  MoveL (T16970) to (106.02, 107.35, 18.1) mm, rotated rx 180 ry 0 rz -180 deg; joints [2.549, 70.013, -35.529, 4.496, -34.567, -3.705]
  Call Extruder 0.1339
  MoveL (T16971) to (109.55, 103.82, 18.1) mm, rotated rx 180 ry 0 rz -180 deg; joints [2.138, 71.113, -37.597, 3.868, -33.577, -3.224]
  Call Extruder 0.01361
  MoveL (T16972) to (109.04, 103.82, 18.1) mm, rotated rx 180 ry 0 rz -180 deg; joints [2.138, 71.113, -37.597, 3.868, -33.577, -3.224]
  Call Extruder 0.11544
  MoveL (T16973) to (106, 106.86, 18.1) mm, rotated rx 180 ry 0 rz -180 deg; joints [2.138, 71.113, -37.597, 3.868, -33.577, -3.224]
  Call Extruder 0.01361
  MoveL (T16974) to (106, 106.35, 18.1) mm, rotated rx 180 ry 0 rz -180 deg; joints [2.086, 71.108, -37.586, 3.773, -33.579, -3.145]
  Call Extruder 0.09619
  MoveL (T16975) to (108.53, 103.82, 18.1) mm, rotated rx 180 ry 0 rz -180 deg; joints [2.086, 71.108, -37.586, 3.773, -33.579, -3.145]
  Call Extruder 0.01361
  MoveL (T16976) to (108.03, 103.82, 18.1) mm, rotated rx 180 ry 0 rz -180 deg; joints [2.086, 71.108, -37.586, 3.773, -33.579, -3.145]
  Call Extruder 0.07694
  MoveL (T16977) to (106, 105.85, 18.1) mm, rotated rx 180 ry 0 rz -180 deg; joints [2.523, 69.937, -35.386, 4.443, -34.632, -3.658]
  Call Extruder 0.01361
  MoveL (T16978) to (106, 105.34, 18.1) mm, rotated rx 180 ry 0 rz -180 deg; joints [2.523, 69.937, -35.386, 4.443, -34.632, -3.658]
  Call Extruder 0.06379
  MoveL (T16979) to (107.68, 103.66, 18.1) mm, rotated rx 180 ry 0 rz -180 deg; joints [2.519, 69.932, -35.375, 4.435, -34.636, -3.651]
  Set speed (45.0 mm/s)
  Call Extruder -1.6
  MoveL (T16980) to (107.68, 103.66, 18.1) mm, rotated rx 180 ry 0 rz -180 deg; joints [2.519, 69.932, -35.375, 4.435, -34.636, -3.651]
  Set speed (120.0 mm/s)
  MoveL (T16981) to (107.68, 103.66, 18.1) mm, rotated rx 180 ry 0 rz -180 deg; joints [2.519, 69.932, -35.375, 4.435, -34.636, -3.651]
  Call Extruder -0.38
  MoveL (T16982) to (106.93, 104.41, 18.1) mm, rotated rx 180 ry 0 rz -180 deg; joints [2.519, 69.932, -35.375, 4.435, -34.636, -3.651]
  Set speed (45.0 mm/s)
  Call Extruder -0.02
  MoveL (T16983) to (106.93, 104.41, 18.1) mm, rotated rx 180 ry 0 rz -180 deg; joints [2.472, 69.926, -35.365, 4.353, -34.639, -3.583]
  Set speed (150.0 mm/s)
  MoveL (T16984) to (106.93, 104.41, 20.1) mm, rotated rx 180 ry 0 rz -180 deg; joints [2.472, 69.926, -35.365, 4.353, -34.639, -3.583]
  MoveL (T16985) to (108.68, 114.32, 20.1) mm, rotated rx 180 ry 0 rz -180 deg; joints [2.033, 71.102, -37.575, 3.678, -33.581, -3.065]
  MoveL (T16986) to (108.68, 114.32, 18.1) mm, rotated rx 180 ry 0 rz -180 deg; joints [2.033, 71.102, -37.575, 3.678, -33.581, -3.065]
  Set speed (40.0 mm/s)
  Call Extruder 2.0
  MoveL (T16987) to (108.68, 114.32, 18.1) mm, rotated rx 180 ry 0 rz -180 deg; joints [1.981, 71.097, -37.565, 3.582, -33.583, -2.986]
  Set speed (25.0 mm/s)
  MoveL (T16988) to (108.68, 114.32, 18.1) mm, rotated rx 180 ry 0 rz -180 deg; joints [1.981, 71.097, -37.565, 3.582, -33.583, -2.986]
  Call Extruder 0.09856
  MoveL (T16989) to (106.08, 116.92, 18.1) mm, rotated rx 180 ry 0 rz -180 deg; joints [1.981, 71.097, -37.565, 3.582, -33.583, -2.986]
  Call Extruder 0.01361
  MoveL (T16990) to (106.08, 116.41, 18.1) mm, rotated rx 180 ry 0 rz -180 deg; joints [1.981, 71.097, -37.565, 3.582, -33.583, -2.986]
  Call Extruder 0.07931
  MoveL (T16991) to (108.17, 114.32, 18.1) mm, rotated rx 180 ry 0 rz -180 deg; joints [2.42, 69.919, -35.353, 4.259, -34.641, -3.506]
  Set speed (45.0 mm/s)
  Call Extruder -1.6
  MoveL (T16992) to (108.17, 114.32, 18.1) mm, rotated rx 180 ry 0 rz -180 deg; joints [2.42, 69.919, -35.353, 4.259, -34.641, -3.506]
  Set speed (120.0 mm/s)
  MoveL (T16993) to (108.17, 114.32, 18.1) mm, rotated rx 180 ry 0 rz -180 deg; joints [2.42, 69.919, -35.353, 4.259, -34.641, -3.506]
  Call Extruder -0.38
  MoveL (T16994) to (107.42, 115.08, 18.1) mm, rotated rx 180 ry 0 rz -180 deg; joints [2.42, 69.919, -35.353, 4.259, -34.641, -3.506]
  Set speed (45.0 mm/s)
  Call Extruder -0.02
  MoveL (T16995) to (107.42, 115.08, 18.1) mm, rotated rx 180 ry 0 rz -180 deg; joints [2.367, 69.913, -35.341, 4.166, -34.643, -3.429]
  Set speed (150.0 mm/s)
  MoveL (T16996) to (107.42, 115.08, 20.1) mm, rotated rx 180 ry 0 rz -180 deg; joints [2.367, 69.913, -35.341, 4.166, -34.643, -3.429]
  MoveL (T16997) to (109.4, 105.47, 20.1) mm, rotated rx 180 ry 0 rz -180 deg; joints [2.367, 69.913, -35.341, 4.166, -34.643, -3.429]
  MoveL (T16998) to (109.4, 105.47, 18.3) mm, rotated rx 180 ry 0 rz -180 deg; joints [2.367, 69.913, -35.341, 4.166, -34.643, -3.429]
  Set speed (40.0 mm/s)
  Call Extruder 2.0
  MoveL (T16999) to (109.4, 105.47, 18.3) mm, rotated rx 180 ry 0 rz -180 deg; joints [1.928, 71.091, -37.555, 3.487, -33.585, -2.906]
  Set speed (31.5 mm/s)
  MoveL (T17000) to (109.4, 105.47, 18.3) mm, rotated rx 180 ry 0 rz -180 deg; joints [1.928, 71.091, -37.555, 3.487, -33.585, -2.906]
  Call Extruder 0.25145
  MoveL (T17001) to (117.65, 105.47, 18.3) mm, rotated rx 180 ry 0 rz -180 deg; joints [1.876, 71.086, -37.545, 3.392, -33.587, -2.827]
  Call Extruder 0.10939
  MoveL (T17002) to (117.65, 109.06, 18.3) mm, rotated rx 180 ry 0 rz -180 deg; joints [1.876, 71.086, -37.545, 3.392, -33.587, -2.827]
  Call Extruder 0.14732
  MoveL (T17003) to (112.81, 109.06, 18.3) mm, rotated rx 180 ry 0 rz -180 deg; joints [1.876, 71.086, -37.545, 3.392, -33.587, -2.827]
  Call Extruder 0.31102
  MoveL (T17004) to (117.47, 118.15, 18.3) mm, rotated rx 180 ry 0 rz -180 deg; joints [2.314, 69.907, -35.33, 4.072, -34.645, -3.352]
  Call Extruder 0.05209
  MoveL (T17005) to (117.47, 119.86, 18.3) mm, rotated rx 180 ry 0 rz -180 deg; joints [2.314, 69.907, -35.33, 4.072, -34.645, -3.352]
  Call Extruder 0.29244
  MoveL (T17006) to (107.87, 119.86, 18.3) mm, rotated rx 180 ry 0 rz -180 deg; joints [2.314, 69.907, -35.33, 4.072, -34.645, -3.352]
  Call Extruder 0.10939
  MoveL (T17007) to (107.87, 116.27, 18.3) mm, rotated rx 180 ry 0 rz -180 deg; joints [2.314, 69.907, -35.33, 4.072, -34.645, -3.352]
  Call Extruder 0.13869
  MoveL (T17008) to (112.42, 116.27, 18.3) mm, rotated rx 180 ry 0 rz -180 deg; joints [2.261, 69.902, -35.319, 3.979, -34.647, -3.275]
  Call Extruder 0.31084
  MoveL (T17009) to (107.78, 107.18, 18.3) mm, rotated rx 180 ry 0 rz -180 deg; joints [2.261, 69.902, -35.319, 3.979, -34.647, -3.275]
  Call Extruder 0.05206
  MoveL (T17010) to (107.78, 105.47, 18.3) mm, rotated rx 180 ry 0 rz -180 deg; joints [1.826, 71.072, -37.519, 3.302, -33.597, -2.751]
  Call Extruder 0.04735
  MoveL (T17011) to (109.34, 105.47, 18.3) mm, rotated rx 180 ry 0 rz -180 deg; joints [1.826, 71.072, -37.519, 3.302, -33.597, -2.751]
  Set speed (150.0 mm/s)
  MoveL (T17012) to (109, 105.88, 18.3) mm, rotated rx 180 ry 0 rz -180 deg; joints [1.826, 71.072, -37.519, 3.302, -33.597, -2.751]
  Set speed (31.5 mm/s)
  MoveL (T17013) to (109, 105.88, 18.3) mm, rotated rx 180 ry 0 rz -180 deg; joints [1.828, 70.917, -37.227, 3.293, -33.734, -2.74]
  Call Extruder 0.25124
  MoveL (T17014) to (117.24, 105.88, 18.3) mm, rotated rx 180 ry 0 rz -180 deg; joints [1.828, 70.917, -37.227, 3.293, -33.734, -2.74]
  Call Extruder 0.08459
  MoveL (T17015) to (117.24, 108.65, 18.3) mm, rotated rx 180 ry 0 rz -180 deg; joints [1.828, 70.917, -37.227, 3.293, -33.734, -2.74]
  Call Extruder 0.1552
  MoveL (T17016) to (112.15, 108.65, 18.3) mm, rotated rx 180 ry 0 rz -180 deg; joints [1.828, 70.917, -37.227, 3.293, -33.734, -2.74]
  Call Extruder 0.32831
  MoveL (T17017) to (117.06, 118.25, 18.3) mm, rotated rx 180 ry 0 rz -180 deg; joints [2.208, 69.896, -35.308, 3.886, -34.649, -3.198]
  Call Extruder 0.0367
  MoveL (T17018) to (117.06, 119.45, 18.3) mm, rotated rx 180 ry 0 rz -180 deg; joints [2.208, 69.896, -35.308, 3.886, -34.649, -3.198]
  Call Extruder 0.26763
  MoveL (T17019) to (108.27, 119.45, 18.3) mm, rotated rx 180 ry 0 rz -180 deg; joints [2.155, 69.89, -35.298, 3.793, -34.651, -3.121]
  Call Extruder 0.08459
  MoveL (T17020) to (108.27, 116.67, 18.3) mm, rotated rx 180 ry 0 rz -180 deg; joints [2.155, 69.89, -35.298, 3.793, -34.651, -3.121]
  Call Extruder 0.14654
  MoveL (T17021) to (113.08, 116.67, 18.3) mm, rotated rx 180 ry 0 rz -180 deg; joints [1.83, 70.762, -36.936, 3.284, -33.87, -2.728]
  Call Extruder 0.32811
  MoveL (T17022) to (108.19, 107.08, 18.3) mm, rotated rx 180 ry 0 rz -180 deg; joints [1.83, 70.762, -36.936, 3.284, -33.87, -2.728]
  Call Extruder 0.03668
  MoveL (T17023) to (108.19, 105.88, 18.3) mm, rotated rx 180 ry 0 rz -180 deg; joints [1.831, 70.608, -36.647, 3.276, -34.005, -2.717]
  Call Extruder 0.02276
  MoveL (T17024) to (108.94, 105.88, 18.3) mm, rotated rx 180 ry 0 rz -180 deg; joints [1.831, 70.608, -36.647, 3.276, -34.005, -2.717]
  Set speed (150.0 mm/s)
  MoveL (T17025) to (108.6, 106.28, 18.3) mm, rotated rx 180 ry 0 rz -180 deg; joints [1.831, 70.608, -36.647, 3.276, -34.005, -2.717]
  Set speed (25.0 mm/s)
  MoveL (T17026) to (108.6, 106.28, 18.3) mm, rotated rx 180 ry 0 rz -180 deg; joints [2.103, 69.885, -35.287, 3.699, -34.653, -3.045]
  Call Extruder 0.25102
  MoveL (T17027) to (116.84, 106.28, 18.3) mm, rotated rx 180 ry 0 rz -180 deg; joints [2.103, 69.885, -35.287, 3.699, -34.653, -3.045]
  Call Extruder 0.05979
  MoveL (T17028) to (116.84, 108.25, 18.3) mm, rotated rx 180 ry 0 rz -180 deg; joints [2.103, 69.885, -35.287, 3.699, -34.653, -3.045]
  Call Extruder 0.16307
  MoveL (T17029) to (111.48, 108.25, 18.3) mm, rotated rx 180 ry 0 rz -180 deg; joints [2.053, 69.88, -35.278, 3.612, -34.655, -2.972]
  Call Extruder 0.3456
  MoveL (T17030) to (116.65, 118.34, 18.3) mm, rotated rx 180 ry 0 rz -180 deg; joints [2.053, 69.88, -35.278, 3.612, -34.655, -2.972]
  Call Extruder 0.02131
  MoveL (T17031) to (116.65, 119.04, 18.3) mm, rotated rx 180 ry 0 rz -180 deg; joints [2.053, 69.88, -35.278, 3.612, -34.655, -2.972]
  Call Extruder 0.24283
  MoveL (T17032) to (108.68, 119.04, 18.3) mm, rotated rx 180 ry 0 rz -180 deg; joints [2.053, 69.88, -35.278, 3.612, -34.655, -2.972]
  Call Extruder 0.05979
  MoveL (T17033) to (108.68, 117.08, 18.3) mm, rotated rx 180 ry 0 rz -180 deg; joints [2.047, 69.886, -35.289, 3.602, -34.649, -2.965]
  Call Extruder 0.15438
  MoveL (T17034) to (113.75, 117.08, 18.3) mm, rotated rx 180 ry 0 rz -180 deg; joints [2.047, 69.886, -35.289, 3.602, -34.649, -2.965]
  Call Extruder 0.34538
  MoveL (T17035) to (108.6, 106.98, 18.3) mm, rotated rx 180 ry 0 rz -180 deg; joints [1.816, 70.502, -36.447, 3.241, -34.097, -2.685]
  Call Extruder 0.01947
  MoveL (T17036) to (108.6, 106.34, 18.3) mm, rotated rx 180 ry 0 rz -180 deg; joints [1.816, 70.502, -36.447, 3.241, -34.097, -2.685]
  Set speed (150.0 mm/s)
  MoveL (T17037) to (108.54, 105.89, 18.3) mm, rotated rx 180 ry 0 rz -180 deg; joints [1.816, 70.502, -36.447, 3.241, -34.097, -2.685]
  Set speed (45.0 mm/s)
  Call Extruder -1.6
  MoveL (T17038) to (108.54, 105.89, 18.3) mm, rotated rx 180 ry 0 rz -180 deg; joints [1.816, 70.502, -36.447, 3.241, -34.097, -2.685]
  Set speed (120.0 mm/s)
  MoveL (T17039) to (108.54, 105.89, 18.3) mm, rotated rx 180 ry 0 rz -180 deg; joints [1.816, 70.502, -36.447, 3.241, -34.097, -2.685]
  Call Extruder -0.38
  MoveL (T17040) to (109.66, 106.33, 18.3) mm, rotated rx 180 ry 0 rz -180 deg; joints [1.816, 70.502, -36.447, 3.241, -34.097, -2.685]
  Set speed (45.0 mm/s)
  Call Extruder -0.02
  MoveL (T17041) to (109.66, 106.33, 18.3) mm, rotated rx 180 ry 0 rz -180 deg; joints [1.816, 70.502, -36.447, 3.241, -34.097, -2.685]
  Set speed (150.0 mm/s)
  MoveL (T17042) to (109.66, 106.33, 20.3) mm, rotated rx 180 ry 0 rz -180 deg; joints [1.816, 70.502, -36.447, 3.241, -34.097, -2.685]
  MoveL (T17043) to (104.34, 103.54, 20.3) mm, rotated rx 180 ry 0 rz -180 deg; joints [1.816, 70.502, -36.447, 3.241, -34.097, -2.685]
  MoveL (T17044) to (104.34, 103.54, 18.3) mm, rotated rx 180 ry 0 rz -180 deg; joints [1.816, 70.502, -36.447, 3.241, -34.097, -2.685]
  Set speed (40.0 mm/s)
  Call Extruder 2.0
  MoveL (T17045) to (104.34, 103.54, 18.3) mm, rotated rx 180 ry 0 rz -180 deg; joints [1.816, 70.502, -36.447, 3.241, -34.097, -2.685]
  Set speed (31.5 mm/s)
  MoveL (T17046) to (104.34, 103.54, 18.3) mm, rotated rx 180 ry 0 rz -180 deg; joints [1.816, 70.502, -36.447, 3.241, -34.097, -2.685]
  Call Extruder 0.52159
  MoveL (T17047) to (121.46, 103.54, 18.3) mm, rotated rx 180 ry 0 rz -180 deg; joints [1.898, 70.28, -36.031, 3.37, -34.296, -2.785]
  Call Extruder 0.54596
  MoveL (T17048) to (121.46, 121.46, 18.3) mm, rotated rx 180 ry 0 rz -180 deg; joints [1.898, 70.28, -36.031, 3.37, -34.296, -2.785]
  Call Extruder 0.54596
  MoveL (T17049) to (103.54, 121.46, 18.3) mm, rotated rx 180 ry 0 rz -180 deg; joints [1.898, 70.28, -36.031, 3.37, -34.296, -2.785]
  Call Extruder 0.54596
  MoveL (T17050) to (103.54, 103.54, 18.3) mm, rotated rx 180 ry 0 rz -180 deg; joints [1.898, 70.28, -36.031, 3.37, -34.296, -2.785]
  Call Extruder 0.02254
  MoveL (T17051) to (104.28, 103.54, 18.3) mm, rotated rx 180 ry 0 rz -180 deg; joints [1.898, 70.28, -36.031, 3.37, -34.296, -2.785]
  Set speed (150.0 mm/s)
  MoveL (T17052) to (103.53, 103.13, 18.3) mm, rotated rx 180 ry 0 rz -180 deg; joints [1.898, 70.28, -36.031, 3.37, -34.296, -2.785]
  Set speed (31.5 mm/s)
  MoveL (T17053) to (103.53, 103.13, 18.3) mm, rotated rx 180 ry 0 rz -180 deg; joints [1.898, 70.28, -36.031, 3.37, -34.296, -2.785]
  Call Extruder 0.55858
  MoveL (T17054) to (121.87, 103.13, 18.3) mm, rotated rx 180 ry 0 rz -180 deg; joints [1.586, 70.545, -36.923, 2.863, -33.655, -2.384]
  Call Extruder 0.57077
  MoveL (T17055) to (121.87, 121.87, 18.3) mm, rotated rx 180 ry 0 rz -180 deg; joints [1.586, 70.778, -36.966, 2.849, -33.845, -2.367]
  Call Extruder 0.57077
  MoveL (T17056) to (103.13, 121.87, 18.3) mm, rotated rx 180 ry 0 rz -180 deg; joints [1.586, 70.778, -36.966, 2.849, -33.845, -2.367]
  Call Extruder 0.57077
  MoveL (T17057) to (103.13, 103.13, 18.3) mm, rotated rx 180 ry 0 rz -180 deg; joints [1.586, 70.778, -36.966, 2.849, -33.845, -2.367]
  Call Extruder 0.01036
  MoveL (T17058) to (103.47, 103.13, 18.3) mm, rotated rx 180 ry 0 rz -180 deg; joints [1.586, 70.778, -36.966, 2.849, -33.845, -2.367]
  Set speed (150.0 mm/s)
  MoveL (T17059) to (102.72, 102.81, 18.3) mm, rotated rx 180 ry 0 rz -180 deg; joints [1.586, 70.778, -36.966, 2.849, -33.845, -2.367]
  Set speed (25.0 mm/s)
  MoveL (T17060) to (102.72, 102.81, 18.3) mm, rotated rx 180 ry 0 rz -180 deg; joints [1.586, 70.778, -36.966, 2.849, -33.845, -2.367]
  Call Extruder 0.00259
  MoveL (T17061) to (102.72, 102.72, 18.3) mm, rotated rx 180 ry 0 rz -180 deg; joints [1.586, 70.778, -36.966, 2.849, -33.845, -2.367]
  Call Extruder 0.59557
  MoveL (T17062) to (122.28, 102.72, 18.3) mm, rotated rx 180 ry 0 rz -180 deg; joints [1.586, 70.778, -36.966, 2.849, -33.845, -2.367]
  Call Extruder 0.59557
  MoveL (T17063) to (122.28, 122.28, 18.3) mm, rotated rx 180 ry 0 rz -180 deg; joints [1.816, 70.153, -35.791, 3.215, -34.404, -2.654]
  Call Extruder 0.59557
  MoveL (T17064) to (102.72, 122.28, 18.3) mm, rotated rx 180 ry 0 rz -180 deg; joints [1.816, 70.153, -35.791, 3.215, -34.404, -2.654]
  Call Extruder 0.59115
  MoveL (T17065) to (102.72, 102.87, 18.3) mm, rotated rx 180 ry 0 rz -180 deg; joints [1.816, 70.153, -35.791, 3.215, -34.404, -2.654]
  Set speed (150.0 mm/s)
  MoveL (T17066) to (102.78, 102.75, 18.3) mm, rotated rx 180 ry 0 rz -180 deg; joints [1.816, 70.153, -35.791, 3.215, -34.404, -2.654]
  Set speed (45.0 mm/s)
  Call Extruder -1.6
  MoveL (T17067) to (102.78, 102.75, 18.3) mm, rotated rx 180 ry 0 rz -180 deg; joints [1.819, 70.136, -35.759, 3.219, -34.419, -2.656]
  Set speed (120.0 mm/s)
  MoveL (T17068) to (102.78, 102.75, 18.3) mm, rotated rx 180 ry 0 rz -180 deg; joints [1.819, 70.136, -35.759, 3.219, -34.419, -2.656]
  Call Extruder -0.05166
  MoveL (T17069) to (102.72, 102.72, 18.3) mm, rotated rx 180 ry 0 rz -180 deg; joints [1.819, 70.136, -35.759, 3.219, -34.419, -2.656]
  Call Extruder -0.32834
  MoveL (T17070) to (103.65, 102.72, 18.3) mm, rotated rx 180 ry 0 rz -180 deg; joints [1.82, 69.997, -35.498, 3.211, -34.541, -2.646]
  Set speed (45.0 mm/s)
  Call Extruder -0.02
  MoveL (T17071) to (103.65, 102.72, 18.3) mm, rotated rx 180 ry 0 rz -180 deg; joints [1.82, 69.997, -35.498, 3.211, -34.541, -2.646]
  Set speed (150.0 mm/s)
  MoveL (T17072) to (103.65, 102.72, 20.3) mm, rotated rx 180 ry 0 rz -180 deg; joints [1.551, 70.727, -36.87, 2.782, -33.888, -2.31]
  MoveL (T17073) to (106.29, 103.84, 20.3) mm, rotated rx 180 ry 0 rz -180 deg; joints [1.551, 70.727, -36.87, 2.782, -33.888, -2.31]
  MoveL (T17074) to (106.29, 103.84, 18.3) mm, rotated rx 180 ry 0 rz -180 deg; joints [1.551, 70.727, -36.87, 2.782, -33.888, -2.31]
  Set speed (40.0 mm/s)
  Call Extruder 2.0
  MoveL (T17075) to (106.29, 103.84, 18.3) mm, rotated rx 180 ry 0 rz -180 deg; joints [1.499, 70.723, -36.863, 2.688, -33.889, -2.232]
  Set speed (31.5 mm/s)
  MoveL (T17076) to (106.29, 103.84, 18.3) mm, rotated rx 180 ry 0 rz -180 deg; joints [1.499, 70.723, -36.863, 2.688, -33.889, -2.232]
  Call Extruder 0.07441
  MoveL (T17077) to (103.84, 103.84, 18.3) mm, rotated rx 180 ry 0 rz -180 deg; joints [1.822, 69.849, -35.221, 3.204, -34.67, -2.636]
  Call Extruder 0.16673
  MoveL (T17078) to (107.71, 107.71, 18.3) mm, rotated rx 180 ry 0 rz -180 deg; joints [1.822, 69.849, -35.221, 3.204, -34.67, -2.636]
  Call Extruder 0.00815
  MoveL (T17079) to (107.84, 107.95, 18.3) mm, rotated rx 180 ry 0 rz -180 deg; joints [1.823, 69.702, -34.944, 3.196, -34.8, -2.625]
  Call Extruder 0.17197
  MoveL (T17080) to (103.84, 111.94, 18.3) mm, rotated rx 180 ry 0 rz -180 deg; joints [1.823, 69.702, -34.944, 3.196, -34.8, -2.625]
  Call Extruder 0.03385
  MoveL (T17081) to (103.84, 113.06, 18.3) mm, rotated rx 180 ry 0 rz -180 deg; joints [1.823, 69.702, -34.944, 3.196, -34.8, -2.625]
  Call Extruder 0.16015
  MoveL (T17082) to (107.56, 116.77, 18.3) mm, rotated rx 180 ry 0 rz -180 deg; joints [1.446, 70.719, -36.855, 2.594, -33.891, -2.154]
  Call Extruder 0.02027
  MoveL (T17083) to (107.56, 117.44, 18.3) mm, rotated rx 180 ry 0 rz -180 deg; joints [1.446, 70.719, -36.855, 2.594, -33.891, -2.154]
  Call Extruder 0.16015
  MoveL (T17084) to (103.84, 121.16, 18.3) mm, rotated rx 180 ry 0 rz -180 deg; joints [1.395, 70.715, -36.848, 2.503, -33.892, -2.078]
  Call Extruder 0.07441
  MoveL (T17085) to (106.29, 121.16, 18.3) mm, rotated rx 180 ry 0 rz -180 deg; joints [1.395, 70.715, -36.848, 2.503, -33.892, -2.078]
  Set speed (45.0 mm/s)
  Call Extruder -1.6
  MoveL (T17086) to (106.29, 121.16, 18.3) mm, rotated rx 180 ry 0 rz -180 deg; joints [1.395, 70.715, -36.848, 2.503, -33.892, -2.078]
  Set speed (120.0 mm/s)
  MoveL (T17087) to (106.29, 121.16, 18.3) mm, rotated rx 180 ry 0 rz -180 deg; joints [1.395, 70.711, -36.84, 2.503, -33.896, -2.078]
  Call Extruder -0.38
  MoveL (T17088) to (105.22, 121.16, 18.3) mm, rotated rx 180 ry 0 rz -180 deg; joints [1.395, 70.711, -36.84, 2.503, -33.896, -2.078]
  Set speed (45.0 mm/s)
  Call Extruder -0.02
  MoveL (T17089) to (105.22, 121.16, 18.3) mm, rotated rx 180 ry 0 rz -180 deg; joints [1.825, 69.556, -34.67, 3.189, -34.928, -2.615]
  Set speed (150.0 mm/s)
  MoveL (T17090) to (105.22, 121.16, 20.3) mm, rotated rx 180 ry 0 rz -180 deg; joints [1.827, 69.411, -34.398, 3.182, -35.055, -2.605]
  MoveL (T17091) to (109.84, 111.88, 20.3) mm, rotated rx 180 ry 0 rz -180 deg; joints [1.827, 69.411, -34.398, 3.182, -35.055, -2.605]
  MoveL (T17092) to (109.84, 111.88, 18.3) mm, rotated rx 180 ry 0 rz -180 deg; joints [1.827, 69.411, -34.398, 3.182, -35.055, -2.605]
  Set speed (40.0 mm/s)
  Call Extruder 2.0
  MoveL (T17093) to (109.84, 111.88, 18.3) mm, rotated rx 180 ry 0 rz -180 deg; joints [1.397, 70.559, -36.554, 2.496, -34.03, -2.069]
  Set speed (31.5 mm/s)
  MoveL (T17094) to (109.84, 111.88, 18.3) mm, rotated rx 180 ry 0 rz -180 deg; joints [1.397, 70.559, -36.554, 2.496, -34.03, -2.069]
  Call Extruder 0.07441
  MoveL (T17095) to (110.95, 114.05, 18.3) mm, rotated rx 180 ry 0 rz -180 deg; joints [1.397, 70.559, -36.554, 2.496, -34.03, -2.069]
  Call Extruder 0.08223
  MoveL (T17096) to (109.04, 115.96, 18.3) mm, rotated rx 180 ry 0 rz -180 deg; joints [1.398, 70.407, -36.269, 2.49, -34.163, -2.061]
  Call Extruder 0.07057
  MoveL (T17097) to (111.36, 115.96, 18.3) mm, rotated rx 180 ry 0 rz -180 deg; joints [1.398, 70.407, -36.269, 2.49, -34.163, -2.061]
  Call Extruder 0.32359
  MoveL (T17098) to (103.84, 108.45, 18.3) mm, rotated rx 180 ry 0 rz -180 deg; joints [1.829, 69.267, -34.127, 3.175, -35.182, -2.596]
  Call Extruder 0.03385
  MoveL (T17099) to (103.84, 107.34, 18.3) mm, rotated rx 180 ry 0 rz -180 deg; joints [1.829, 69.267, -34.127, 3.175, -35.182, -2.596]
  Call Extruder 0.15054
  MoveL (T17100) to (107.34, 103.84, 18.3) mm, rotated rx 180 ry 0 rz -180 deg; joints [1.83, 69.124, -33.858, 3.168, -35.308, -2.586]
  Call Extruder 0.03385
  MoveL (T17101) to (108.45, 103.84, 18.3) mm, rotated rx 180 ry 0 rz -180 deg; joints [1.83, 69.124, -33.858, 3.168, -35.308, -2.586]
  Call Extruder 0.05679
  MoveL (T17102) to (109.77, 105.16, 18.3) mm, rotated rx 180 ry 0 rz -180 deg; joints [1.83, 69.124, -33.858, 3.168, -35.308, -2.586]
  Call Extruder 0.02614
  MoveL (T17103) to (110.63, 105.16, 18.3) mm, rotated rx 180 ry 0 rz -180 deg; joints [1.83, 69.124, -33.858, 3.168, -35.308, -2.586]
  Call Extruder 0.05679
  MoveL (T17104) to (111.94, 103.84, 18.3) mm, rotated rx 180 ry 0 rz -180 deg; joints [1.399, 70.257, -35.986, 2.484, -34.295, -2.053]
  Call Extruder 0.03385
  MoveL (T17105) to (113.06, 103.84, 18.3) mm, rotated rx 180 ry 0 rz -180 deg; joints [1.399, 70.257, -35.986, 2.484, -34.295, -2.053]
  Call Extruder 0.05679
  MoveL (T17106) to (114.37, 105.16, 18.3) mm, rotated rx 180 ry 0 rz -180 deg; joints [1.399, 70.257, -35.986, 2.484, -34.295, -2.053]
  Call Extruder 0.02614
  MoveL (T17107) to (115.23, 105.16, 18.3) mm, rotated rx 180 ry 0 rz -180 deg; joints [1.401, 70.107, -35.706, 2.478, -34.427, -2.044]
  Call Extruder 0.05679
  MoveL (T17108) to (116.55, 103.84, 18.3) mm, rotated rx 180 ry 0 rz -180 deg; joints [1.401, 70.107, -35.706, 2.478, -34.427, -2.044]
  Call Extruder 0.03385
  MoveL (T17109) to (117.66, 103.84, 18.3) mm, rotated rx 180 ry 0 rz -180 deg; joints [1.832, 68.981, -33.59, 3.161, -35.433, -2.576]
  Call Extruder 0.15054
  MoveL (T17110) to (121.16, 107.34, 18.3) mm, rotated rx 180 ry 0 rz -180 deg; joints [1.832, 68.981, -33.59, 3.161, -35.433, -2.576]
  Call Extruder 0.03385
  MoveL (T17111) to (121.16, 108.45, 18.3) mm, rotated rx 180 ry 0 rz -180 deg; joints [1.834, 68.84, -33.323, 3.154, -35.557, -2.567]
  Call Extruder 0.23679
  MoveL (T17112) to (115.66, 113.95, 18.3) mm, rotated rx 180 ry 0 rz -180 deg; joints [1.402, 69.958, -35.426, 2.472, -34.557, -2.036]
  Call Extruder 0.10426
  MoveL (T17113) to (114.1, 110.9, 18.3) mm, rotated rx 180 ry 0 rz -180 deg; joints [1.402, 69.958, -35.426, 2.472, -34.557, -2.036]
  Call Extruder 0.06615
  MoveL (T17114) to (115.64, 109.36, 18.3) mm, rotated rx 180 ry 0 rz -180 deg; joints [1.402, 69.958, -35.426, 2.472, -34.557, -2.036]
  Call Extruder 0.05076
  MoveL (T17115) to (113.97, 109.36, 18.3) mm, rotated rx 180 ry 0 rz -180 deg; joints [1.403, 69.811, -35.149, 2.466, -34.687, -2.028]
  Call Extruder 0.30958
  MoveL (T17116) to (121.16, 116.55, 18.3) mm, rotated rx 180 ry 0 rz -180 deg; joints [1.403, 69.811, -35.149, 2.466, -34.687, -2.028]
  Call Extruder 0.03385
  MoveL (T17117) to (121.16, 117.66, 18.3) mm, rotated rx 180 ry 0 rz -180 deg; joints [1.403, 69.811, -35.149, 2.466, -34.687, -2.028]
  Call Extruder 0.15054
  MoveL (T17118) to (117.66, 121.16, 18.3) mm, rotated rx 180 ry 0 rz -180 deg; joints [1.814, 68.753, -33.16, 3.114, -35.633, -2.532]
  Call Extruder 0.03385
  MoveL (T17119) to (116.55, 121.16, 18.3) mm, rotated rx 180 ry 0 rz -180 deg; joints [1.814, 68.753, -33.16, 3.114, -35.633, -2.532]
  Call Extruder 0.04278
  MoveL (T17120) to (115.56, 120.16, 18.3) mm, rotated rx 180 ry 0 rz -180 deg; joints [1.814, 68.753, -33.16, 3.114, -35.633, -2.532]
  Call Extruder 0.04595
  MoveL (T17121) to (114.05, 120.16, 18.3) mm, rotated rx 180 ry 0 rz -180 deg; joints [1.814, 68.753, -33.16, 3.114, -35.633, -2.532]
  Call Extruder 0.04278
  MoveL (T17122) to (113.06, 121.16, 18.3) mm, rotated rx 180 ry 0 rz -180 deg; joints [1.788, 68.68, -33.024, 3.065, -35.695, -2.49]
  Call Extruder 0.03385
  MoveL (T17123) to (111.94, 121.16, 18.3) mm, rotated rx 180 ry 0 rz -180 deg; joints [1.788, 68.68, -33.024, 3.065, -35.695, -2.49]
  Call Extruder 0.04278
  MoveL (T17124) to (110.95, 120.16, 18.3) mm, rotated rx 180 ry 0 rz -180 deg; joints [1.788, 68.68, -33.024, 3.065, -35.695, -2.49]
  Call Extruder 0.04595
  MoveL (T17125) to (109.44, 120.16, 18.3) mm, rotated rx 180 ry 0 rz -180 deg; joints [1.788, 68.68, -33.024, 3.065, -35.695, -2.49]
  Call Extruder 0.04278
  MoveL (T17126) to (108.45, 121.16, 18.3) mm, rotated rx 180 ry 0 rz -180 deg; joints [1.404, 69.664, -34.873, 2.46, -34.816, -2.02]
  Call Extruder 0.03385
  MoveL (T17127) to (107.34, 121.16, 18.3) mm, rotated rx 180 ry 0 rz -180 deg; joints [1.404, 69.664, -34.873, 2.46, -34.816, -2.02]
  Call Extruder 0.15054
  MoveL (T17128) to (103.84, 117.66, 18.3) mm, rotated rx 180 ry 0 rz -180 deg; joints [1.406, 69.519, -34.599, 2.455, -34.944, -2.013]
  Call Extruder 0.03385
  MoveL (T17129) to (103.84, 116.55, 18.3) mm, rotated rx 180 ry 0 rz -180 deg; joints [1.406, 69.519, -34.599, 2.455, -34.944, -2.013]
  Call Extruder 0.23899
  MoveL (T17130) to (109.39, 111, 18.3) mm, rotated rx 180 ry 0 rz -180 deg; joints [1.406, 69.519, -34.599, 2.455, -34.944, -2.013]
  Call Extruder 0.07441
  MoveL (T17131) to (108.28, 108.83, 18.3) mm, rotated rx 180 ry 0 rz -180 deg; joints [1.762, 68.608, -32.888, 3.017, -35.757, -2.449]
  Set speed (45.0 mm/s)
  Call Extruder -1.6
  MoveL (T17132) to (108.28, 108.83, 18.3) mm, rotated rx 180 ry 0 rz -180 deg; joints [1.762, 68.608, -32.888, 3.017, -35.757, -2.449]
  Set speed (120.0 mm/s)
  MoveL (T17133) to (108.28, 108.83, 18.3) mm, rotated rx 180 ry 0 rz -180 deg; joints [1.762, 68.608, -32.888, 3.017, -35.757, -2.449]
  Call Extruder -0.38
  MoveL (T17134) to (108.77, 109.78, 18.3) mm, rotated rx 180 ry 0 rz -180 deg; joints [1.737, 68.536, -32.754, 2.968, -35.819, -2.408]
  Set speed (45.0 mm/s)
  Call Extruder -0.02
  MoveL (T17135) to (108.77, 109.78, 18.3) mm, rotated rx 180 ry 0 rz -180 deg; joints [1.737, 68.536, -32.754, 2.968, -35.819, -2.408]
  Set speed (150.0 mm/s)
  MoveL (T17136) to (108.77, 109.78, 20.3) mm, rotated rx 180 ry 0 rz -180 deg; joints [1.737, 68.536, -32.754, 2.968, -35.819, -2.408]
  MoveL (T17137) to (118.71, 103.84, 20.3) mm, rotated rx 180 ry 0 rz -180 deg; joints [1.737, 68.536, -32.754, 2.968, -35.819, -2.408]
  MoveL (T17138) to (118.71, 103.84, 18.3) mm, rotated rx 180 ry 0 rz -180 deg; joints [1.407, 69.374, -34.327, 2.449, -35.071, -2.005]
  Set speed (40.0 mm/s)
  Call Extruder 2.0
  MoveL (T17139) to (118.71, 103.84, 18.3) mm, rotated rx 180 ry 0 rz -180 deg; joints [1.407, 69.374, -34.327, 2.449, -35.071, -2.005]
  Set speed (31.5 mm/s)
  MoveL (T17140) to (118.71, 103.84, 18.3) mm, rotated rx 180 ry 0 rz -180 deg; joints [1.408, 69.23, -34.056, 2.444, -35.198, -1.997]
  Call Extruder 0.07441
  MoveL (T17141) to (121.16, 103.84, 18.3) mm, rotated rx 180 ry 0 rz -180 deg; joints [1.408, 69.23, -34.056, 2.444, -35.198, -1.997]
  Call Extruder 0.13782
  MoveL (T17142) to (117.96, 107.04, 18.3) mm, rotated rx 180 ry 0 rz -180 deg; joints [1.711, 68.464, -32.618, 2.92, -35.881, -2.366]
  Call Extruder 0.05185
  MoveL (T17143) to (117.96, 108.75, 18.3) mm, rotated rx 180 ry 0 rz -180 deg; joints [1.711, 68.464, -32.618, 2.92, -35.881, -2.366]
  Call Extruder 0.13782
  MoveL (T17144) to (121.16, 111.94, 18.3) mm, rotated rx 180 ry 0 rz -180 deg; joints [1.711, 68.464, -32.618, 2.92, -35.881, -2.366]
  Call Extruder 0.03385
  MoveL (T17145) to (121.16, 113.06, 18.3) mm, rotated rx 180 ry 0 rz -180 deg; joints [1.685, 68.393, -32.484, 2.872, -35.943, -2.326]
  Call Extruder 0.16962
  MoveL (T17146) to (117.22, 116.99, 18.3) mm, rotated rx 180 ry 0 rz -180 deg; joints [1.685, 68.393, -32.484, 2.872, -35.943, -2.326]
  Call Extruder 0.01582
  MoveL (T17147) to (117.45, 117.45, 18.3) mm, rotated rx 180 ry 0 rz -180 deg; joints [1.685, 68.393, -32.484, 2.872, -35.943, -2.326]
  Call Extruder 0.15942
  MoveL (T17148) to (121.16, 121.16, 18.3) mm, rotated rx 180 ry 0 rz -180 deg; joints [1.41, 69.087, -33.788, 2.439, -35.324, -1.99]
  Call Extruder 0.07441
  MoveL (T17149) to (118.71, 121.16, 18.3) mm, rotated rx 180 ry 0 rz -180 deg; joints [1.41, 69.087, -33.788, 2.439, -35.324, -1.99]
  Set speed (45.0 mm/s)
  Call Extruder -1.6
  MoveL (T17150) to (118.71, 121.16, 18.3) mm, rotated rx 180 ry 0 rz -180 deg; joints [1.41, 69.087, -33.788, 2.439, -35.324, -1.99]
  Set speed (120.0 mm/s)
  MoveL (T17151) to (118.71, 121.16, 18.3) mm, rotated rx 180 ry 0 rz -180 deg; joints [1.411, 68.944, -33.52, 2.433, -35.448, -1.983]
  Call Extruder -0.38
  MoveL (T17152) to (119.78, 121.16, 18.3) mm, rotated rx 180 ry 0 rz -180 deg; joints [1.411, 68.944, -33.52, 2.433, -35.448, -1.983]
  Set speed (45.0 mm/s)
  Call Extruder -0.02
  MoveL (T17153) to (119.78, 121.16, 18.3) mm, rotated rx 180 ry 0 rz -180 deg; joints [1.846, 67.87, -31.502, 3.11, -36.408, -2.504]
  Set speed (150.0 mm/s)
  MoveL (T17154) to (119.78, 121.16, 20.3) mm, rotated rx 180 ry 0 rz -180 deg; joints [1.846, 67.87, -31.502, 3.11, -36.408, -2.504]
  MoveL (T17155) to (109.4, 105.47, 20.3) mm, rotated rx 180 ry 0 rz -180 deg; joints [1.846, 67.87, -31.502, 3.11, -36.408, -2.504]
  MoveL (T17156) to (109.4, 105.47, 18.5) mm, rotated rx 180 ry 0 rz -180 deg; joints [1.847, 67.735, -31.248, 3.105, -36.527, -2.496]
  Set speed (40.0 mm/s)
  Call Extruder 2.0
  MoveL (T17157) to (109.4, 105.47, 18.5) mm, rotated rx 180 ry 0 rz -180 deg; joints [1.847, 67.735, -31.248, 3.105, -36.527, -2.496]
  Set speed (31.6 mm/s)
  MoveL (T17158) to (109.4, 105.47, 18.5) mm, rotated rx 180 ry 0 rz -180 deg; joints [1.847, 67.735, -31.248, 3.105, -36.527, -2.496]
  Call Extruder 0.25145
  MoveL (T17159) to (117.65, 105.47, 18.5) mm, rotated rx 180 ry 0 rz -180 deg; joints [1.412, 68.803, -33.255, 2.428, -35.573, -1.975]
  Call Extruder 0.10939
  MoveL (T17160) to (117.65, 109.06, 18.5) mm, rotated rx 180 ry 0 rz -180 deg; joints [1.412, 68.803, -33.255, 2.428, -35.573, -1.975]
  Call Extruder 0.14732
  MoveL (T17161) to (112.81, 109.06, 18.5) mm, rotated rx 180 ry 0 rz -180 deg; joints [1.414, 68.662, -32.99, 2.423, -35.696, -1.968]
  Call Extruder 0.31102
  MoveL (T17162) to (117.47, 118.15, 18.5) mm, rotated rx 180 ry 0 rz -180 deg; joints [1.849, 67.6, -30.994, 3.099, -36.646, -2.487]
  Call Extruder 0.05209
  MoveL (T17163) to (117.47, 119.86, 18.5) mm, rotated rx 180 ry 0 rz -180 deg; joints [1.849, 67.6, -30.994, 3.099, -36.646, -2.487]
  Call Extruder 0.29244
  MoveL (T17164) to (107.87, 119.86, 18.5) mm, rotated rx 180 ry 0 rz -180 deg; joints [1.851, 67.465, -30.742, 3.093, -36.764, -2.479]
  Call Extruder 0.10939
  MoveL (T17165) to (107.87, 116.27, 18.5) mm, rotated rx 180 ry 0 rz -180 deg; joints [1.415, 68.522, -32.727, 2.418, -35.819, -1.961]
  Call Extruder 0.13869
  MoveL (T17166) to (112.42, 116.27, 18.5) mm, rotated rx 180 ry 0 rz -180 deg; joints [1.415, 68.522, -32.727, 2.418, -35.819, -1.961]
  Call Extruder 0.31084
  MoveL (T17167) to (107.78, 107.18, 18.5) mm, rotated rx 180 ry 0 rz -180 deg; joints [1.415, 68.522, -32.727, 2.418, -35.819, -1.961]
  Call Extruder 0.05206
  MoveL (T17168) to (107.78, 105.47, 18.5) mm, rotated rx 180 ry 0 rz -180 deg; joints [1.416, 68.383, -32.466, 2.413, -35.941, -1.954]
  Call Extruder 0.04735
  MoveL (T17169) to (109.34, 105.47, 18.5) mm, rotated rx 180 ry 0 rz -180 deg; joints [1.416, 68.383, -32.466, 2.413, -35.941, -1.954]
  Set speed (150.0 mm/s)
  MoveL (T17170) to (109, 105.88, 18.5) mm, rotated rx 180 ry 0 rz -180 deg; joints [1.416, 68.383, -32.466, 2.413, -35.941, -1.954]
  Set speed (31.6 mm/s)
  MoveL (T17171) to (109, 105.88, 18.5) mm, rotated rx 180 ry 0 rz -180 deg; joints [1.416, 68.383, -32.466, 2.413, -35.941, -1.954]
  Call Extruder 0.25124
  MoveL (T17172) to (117.24, 105.88, 18.5) mm, rotated rx 180 ry 0 rz -180 deg; joints [1.852, 67.332, -30.491, 3.088, -36.881, -2.471]
  Call Extruder 0.08459
  MoveL (T17173) to (117.24, 108.65, 18.5) mm, rotated rx 180 ry 0 rz -180 deg; joints [1.852, 67.332, -30.491, 3.088, -36.881, -2.471]
  Call Extruder 0.1552
  MoveL (T17174) to (112.15, 108.65, 18.5) mm, rotated rx 180 ry 0 rz -180 deg; joints [1.852, 67.332, -30.491, 3.088, -36.881, -2.471]
  Call Extruder 0.32831
  MoveL (T17175) to (117.06, 118.25, 18.5) mm, rotated rx 180 ry 0 rz -180 deg; joints [1.852, 67.332, -30.491, 3.088, -36.881, -2.471]
  Call Extruder 0.0367
  MoveL (T17176) to (117.06, 119.45, 18.5) mm, rotated rx 180 ry 0 rz -180 deg; joints [1.854, 67.199, -30.242, 3.082, -36.997, -2.462]
  Call Extruder 0.26763
  MoveL (T17177) to (108.27, 119.45, 18.5) mm, rotated rx 180 ry 0 rz -180 deg; joints [1.854, 67.199, -30.242, 3.082, -36.997, -2.462]
  Call Extruder 0.08459
  MoveL (T17178) to (108.27, 116.67, 18.5) mm, rotated rx 180 ry 0 rz -180 deg; joints [1.854, 67.199, -30.242, 3.082, -36.997, -2.462]
  Call Extruder 0.14654
  MoveL (T17179) to (113.08, 116.67, 18.5) mm, rotated rx 180 ry 0 rz -180 deg; joints [1.854, 67.199, -30.242, 3.082, -36.997, -2.462]
  Call Extruder 0.32811
  MoveL (T17180) to (108.19, 107.08, 18.5) mm, rotated rx 180 ry 0 rz -180 deg; joints [1.417, 68.245, -32.206, 2.408, -36.063, -1.947]
  Call Extruder 0.03668
  MoveL (T17181) to (108.19, 105.88, 18.5) mm, rotated rx 180 ry 0 rz -180 deg; joints [1.417, 68.245, -32.206, 2.408, -36.063, -1.947]
  Call Extruder 0.02276
  MoveL (T17182) to (108.94, 105.88, 18.5) mm, rotated rx 180 ry 0 rz -180 deg; joints [1.419, 68.107, -31.948, 2.404, -36.184, -1.94]
  Set speed (150.0 mm/s)
  MoveL (T17183) to (108.6, 106.28, 18.5) mm, rotated rx 180 ry 0 rz -180 deg; joints [1.419, 68.107, -31.948, 2.404, -36.184, -1.94]
  Set speed (25.0 mm/s)
  MoveL (T17184) to (108.6, 106.28, 18.5) mm, rotated rx 180 ry 0 rz -180 deg; joints [1.419, 68.107, -31.948, 2.404, -36.184, -1.94]
  Call Extruder 0.25102
  MoveL (T17185) to (116.84, 106.28, 18.5) mm, rotated rx 180 ry 0 rz -180 deg; joints [1.856, 67.067, -29.994, 3.077, -37.113, -2.454]
  Call Extruder 0.05979
  MoveL (T17186) to (116.84, 108.25, 18.5) mm, rotated rx 180 ry 0 rz -180 deg; joints [1.856, 67.067, -29.994, 3.077, -37.113, -2.454]
  Call Extruder 0.16307
  MoveL (T17187) to (111.48, 108.25, 18.5) mm, rotated rx 180 ry 0 rz -180 deg; joints [1.856, 67.067, -29.994, 3.077, -37.113, -2.454]
  Call Extruder 0.3456
  MoveL (T17188) to (116.65, 118.34, 18.5) mm, rotated rx 180 ry 0 rz -180 deg; joints [1.858, 66.936, -29.747, 3.071, -37.229, -2.446]
  Call Extruder 0.02131
  MoveL (T17189) to (116.65, 119.04, 18.5) mm, rotated rx 180 ry 0 rz -180 deg; joints [1.858, 66.936, -29.747, 3.071, -37.229, -2.446]
  Call Extruder 0.24283
  MoveL (T17190) to (108.68, 119.04, 18.5) mm, rotated rx 180 ry 0 rz -180 deg; joints [1.858, 66.936, -29.747, 3.071, -37.229, -2.446]
  Call Extruder 0.05979
  MoveL (T17191) to (108.68, 117.08, 18.5) mm, rotated rx 180 ry 0 rz -180 deg; joints [1.42, 67.971, -31.691, 2.399, -36.304, -1.934]
  Call Extruder 0.15438
  MoveL (T17192) to (113.75, 117.08, 18.5) mm, rotated rx 180 ry 0 rz -180 deg; joints [1.42, 67.971, -31.691, 2.399, -36.304, -1.934]
  Call Extruder 0.34538
  MoveL (T17193) to (108.6, 106.98, 18.5) mm, rotated rx 180 ry 0 rz -180 deg; joints [1.42, 67.971, -31.691, 2.399, -36.304, -1.934]
  Call Extruder 0.01947
  MoveL (T17194) to (108.6, 106.34, 18.5) mm, rotated rx 180 ry 0 rz -180 deg; joints [1.42, 67.971, -31.691, 2.399, -36.304, -1.934]
  Set speed (150.0 mm/s)
  MoveL (T17195) to (108.54, 105.89, 18.5) mm, rotated rx 180 ry 0 rz -180 deg; joints [1.421, 67.834, -31.435, 2.394, -36.423, -1.927]
  Set speed (45.0 mm/s)
  Call Extruder -1.6
  MoveL (T17196) to (108.54, 105.89, 18.5) mm, rotated rx 180 ry 0 rz -180 deg; joints [1.421, 67.834, -31.435, 2.394, -36.423, -1.927]
  Set speed (120.0 mm/s)
  MoveL (T17197) to (108.54, 105.89, 18.5) mm, rotated rx 180 ry 0 rz -180 deg; joints [1.858, 66.808, -29.506, 3.064, -37.341, -2.437]
  Call Extruder -0.38
  MoveL (T17198) to (109.66, 106.33, 18.5) mm, rotated rx 180 ry 0 rz -180 deg; joints [1.858, 66.808, -29.506, 3.064, -37.341, -2.437]
  Set speed (45.0 mm/s)
  Call Extruder -0.02
  MoveL (T17199) to (109.66, 106.33, 18.5) mm, rotated rx 180 ry 0 rz -180 deg; joints [1.857, 66.798, -29.489, 3.061, -37.349, -2.434]
  Set speed (150.0 mm/s)
  MoveL (T17200) to (109.66, 106.33, 20.5) mm, rotated rx 180 ry 0 rz -180 deg; joints [1.857, 66.798, -29.489, 3.061, -37.349, -2.434]
  MoveL (T17201) to (104.34, 103.54, 20.5) mm, rotated rx 180 ry 0 rz -180 deg; joints [1.833, 66.738, -29.375, 3.019, -37.401, -2.399]
  MoveL (T17202) to (104.34, 103.54, 18.5) mm, rotated rx 180 ry 0 rz -180 deg; joints [1.833, 66.738, -29.375, 3.019, -37.401, -2.399]
  Set speed (40.0 mm/s)
  Call Extruder 2.0
  MoveL (T17203) to (104.34, 103.54, 18.5) mm, rotated rx 180 ry 0 rz -180 deg; joints [1.423, 67.699, -31.181, 2.39, -36.542, -1.921]
  Set speed (31.6 mm/s)
  MoveL (T17204) to (104.34, 103.54, 18.5) mm, rotated rx 180 ry 0 rz -180 deg; joints [1.423, 67.699, -31.181, 2.39, -36.542, -1.921]
  Call Extruder 0.52159
  MoveL (T17205) to (121.46, 103.54, 18.5) mm, rotated rx 180 ry 0 rz -180 deg; joints [1.423, 67.699, -31.181, 2.39, -36.542, -1.921]
  Call Extruder 0.54596
  MoveL (T17206) to (121.46, 121.46, 18.5) mm, rotated rx 180 ry 0 rz -180 deg; joints [1.424, 67.564, -30.928, 2.386, -36.66, -1.914]
  Call Extruder 0.54596
  MoveL (T17207) to (103.54, 121.46, 18.5) mm, rotated rx 180 ry 0 rz -180 deg; joints [1.424, 67.564, -30.928, 2.386, -36.66, -1.914]
  Call Extruder 0.54596
  MoveL (T17208) to (103.54, 103.54, 18.5) mm, rotated rx 180 ry 0 rz -180 deg; joints [1.424, 67.564, -30.928, 2.386, -36.66, -1.914]
  Call Extruder 0.02254
  MoveL (T17209) to (104.28, 103.54, 18.5) mm, rotated rx 180 ry 0 rz -180 deg; joints [1.807, 66.671, -29.249, 2.972, -37.459, -2.36]
  Set speed (150.0 mm/s)
  MoveL (T17210) to (103.53, 103.13, 18.5) mm, rotated rx 180 ry 0 rz -180 deg; joints [1.807, 66.671, -29.249, 2.972, -37.459, -2.36]
  Set speed (31.6 mm/s)
  MoveL (T17211) to (103.53, 103.13, 18.5) mm, rotated rx 180 ry 0 rz -180 deg; joints [1.807, 66.671, -29.249, 2.972, -37.459, -2.36]
  Call Extruder 0.55858
  MoveL (T17212) to (121.87, 103.13, 18.5) mm, rotated rx 180 ry 0 rz -180 deg; joints [1.781, 66.604, -29.124, 2.926, -37.516, -2.322]
  Call Extruder 0.57077
  MoveL (T17213) to (121.87, 121.87, 18.5) mm, rotated rx 180 ry 0 rz -180 deg; joints [1.781, 66.604, -29.124, 2.926, -37.516, -2.322]
  Call Extruder 0.57077
  MoveL (T17214) to (103.13, 121.87, 18.5) mm, rotated rx 180 ry 0 rz -180 deg; joints [1.781, 66.604, -29.124, 2.926, -37.516, -2.322]
  Call Extruder 0.57077
  MoveL (T17215) to (103.13, 103.13, 18.5) mm, rotated rx 180 ry 0 rz -180 deg; joints [1.781, 66.604, -29.124, 2.926, -37.516, -2.322]
  Call Extruder 0.01036
  MoveL (T17216) to (103.47, 103.13, 18.5) mm, rotated rx 180 ry 0 rz -180 deg; joints [1.425, 67.43, -30.676, 2.381, -36.778, -1.908]
  Set speed (150.0 mm/s)
  MoveL (T17217) to (102.72, 102.81, 18.5) mm, rotated rx 180 ry 0 rz -180 deg; joints [1.425, 67.43, -30.676, 2.381, -36.778, -1.908]
  Set speed (25.0 mm/s)
  MoveL (T17218) to (102.72, 102.81, 18.5) mm, rotated rx 180 ry 0 rz -180 deg; joints [1.427, 67.297, -30.426, 2.377, -36.895, -1.901]
  Call Extruder 0.00259
  MoveL (T17219) to (102.72, 102.72, 18.5) mm, rotated rx 180 ry 0 rz -180 deg; joints [1.427, 67.297, -30.426, 2.377, -36.895, -1.901]
  Call Extruder 0.59557
  MoveL (T17220) to (122.28, 102.72, 18.5) mm, rotated rx 180 ry 0 rz -180 deg; joints [1.755, 66.537, -28.998, 2.879, -37.574, -2.283]
  Call Extruder 0.59557
  MoveL (T17221) to (122.28, 122.28, 18.5) mm, rotated rx 180 ry 0 rz -180 deg; joints [1.755, 66.537, -28.998, 2.879, -37.574, -2.283]
  Call Extruder 0.59557
  MoveL (T17222) to (102.72, 122.28, 18.5) mm, rotated rx 180 ry 0 rz -180 deg; joints [1.729, 66.471, -28.874, 2.833, -37.631, -2.244]
  Call Extruder 0.59115
  MoveL (T17223) to (102.72, 102.87, 18.5) mm, rotated rx 180 ry 0 rz -180 deg; joints [1.729, 66.471, -28.874, 2.833, -37.631, -2.244]
  Set speed (150.0 mm/s)
  MoveL (T17224) to (102.78, 102.75, 18.5) mm, rotated rx 180 ry 0 rz -180 deg; joints [1.729, 66.471, -28.874, 2.833, -37.631, -2.244]
  Set speed (45.0 mm/s)
  Call Extruder -1.6
  MoveL (T17225) to (102.78, 102.75, 18.5) mm, rotated rx 180 ry 0 rz -180 deg; joints [1.428, 67.164, -30.176, 2.373, -37.012, -1.895]
  Set speed (120.0 mm/s)
  MoveL (T17226) to (102.78, 102.75, 18.5) mm, rotated rx 180 ry 0 rz -180 deg; joints [1.428, 67.164, -30.176, 2.373, -37.012, -1.895]
  Call Extruder -0.05166
  MoveL (T17227) to (102.72, 102.72, 18.5) mm, rotated rx 180 ry 0 rz -180 deg; joints [1.429, 67.032, -29.929, 2.369, -37.127, -1.889]
  Call Extruder -0.32834
  MoveL (T17228) to (103.65, 102.72, 18.5) mm, rotated rx 180 ry 0 rz -180 deg; joints [1.429, 67.032, -29.929, 2.369, -37.127, -1.889]
  Set speed (45.0 mm/s)
  Call Extruder -0.02
  MoveL (T17229) to (103.65, 102.72, 18.5) mm, rotated rx 180 ry 0 rz -180 deg; joints [1.429, 67.032, -29.929, 2.369, -37.127, -1.889]
  Set speed (150.0 mm/s)
  MoveL (T17230) to (103.65, 102.72, 20.5) mm, rotated rx 180 ry 0 rz -180 deg; joints [1.703, 66.404, -28.749, 2.787, -37.688, -2.206]
  MoveL (T17231) to (106.29, 103.84, 20.5) mm, rotated rx 180 ry 0 rz -180 deg; joints [1.703, 66.404, -28.749, 2.787, -37.688, -2.206]
  MoveL (T17232) to (106.29, 103.84, 18.5) mm, rotated rx 180 ry 0 rz -180 deg; joints [1.703, 66.404, -28.749, 2.787, -37.688, -2.206]
  Set speed (40.0 mm/s)
  Call Extruder 2.0
  MoveL (T17233) to (106.29, 103.84, 18.5) mm, rotated rx 180 ry 0 rz -180 deg; joints [1.677, 66.338, -28.624, 2.74, -37.745, -2.168]
  Set speed (31.6 mm/s)
  MoveL (T17234) to (106.29, 103.84, 18.5) mm, rotated rx 180 ry 0 rz -180 deg; joints [1.677, 66.338, -28.624, 2.74, -37.745, -2.168]
  Call Extruder 0.07441
  MoveL (T17235) to (103.84, 103.84, 18.5) mm, rotated rx 180 ry 0 rz -180 deg; joints [1.677, 66.338, -28.624, 2.74, -37.745, -2.168]
  Call Extruder 0.16673
  MoveL (T17236) to (107.71, 107.71, 18.5) mm, rotated rx 180 ry 0 rz -180 deg; joints [1.431, 66.901, -29.682, 2.365, -37.243, -1.883]
  Call Extruder 0.00815
  MoveL (T17237) to (107.84, 107.95, 18.5) mm, rotated rx 180 ry 0 rz -180 deg; joints [1.431, 66.901, -29.682, 2.365, -37.243, -1.883]
  Call Extruder 0.17197
  MoveL (T17238) to (103.84, 111.94, 18.5) mm, rotated rx 180 ry 0 rz -180 deg; joints [1.432, 66.77, -29.437, 2.361, -37.357, -1.877]
  Call Extruder 0.03385
  MoveL (T17239) to (103.84, 113.06, 18.5) mm, rotated rx 180 ry 0 rz -180 deg; joints [1.432, 66.77, -29.437, 2.361, -37.357, -1.877]
  Call Extruder 0.16015
  MoveL (T17240) to (107.56, 116.77, 18.5) mm, rotated rx 180 ry 0 rz -180 deg; joints [1.649, 66.276, -28.507, 2.692, -37.799, -2.128]
  Call Extruder 0.02027
  MoveL (T17241) to (107.56, 117.44, 18.5) mm, rotated rx 180 ry 0 rz -180 deg; joints [1.649, 66.276, -28.507, 2.692, -37.799, -2.128]
  Call Extruder 0.16015
  MoveL (T17242) to (103.84, 121.16, 18.5) mm, rotated rx 180 ry 0 rz -180 deg; joints [1.596, 66.271, -28.498, 2.605, -37.801, -2.059]
  Call Extruder 0.07441
  MoveL (T17243) to (106.29, 121.16, 18.5) mm, rotated rx 180 ry 0 rz -180 deg; joints [1.596, 66.271, -28.498, 2.605, -37.801, -2.059]
  Set speed (45.0 mm/s)
  Call Extruder -1.6
  MoveL (T17244) to (106.29, 121.16, 18.5) mm, rotated rx 180 ry 0 rz -180 deg; joints [1.433, 66.64, -29.193, 2.357, -37.471, -1.871]
  Set speed (120.0 mm/s)
  MoveL (T17245) to (106.29, 121.16, 18.5) mm, rotated rx 180 ry 0 rz -180 deg; joints [1.433, 66.64, -29.193, 2.357, -37.471, -1.871]
  Call Extruder -0.38
  MoveL (T17246) to (105.22, 121.16, 18.5) mm, rotated rx 180 ry 0 rz -180 deg; joints [1.435, 66.511, -28.949, 2.353, -37.585, -1.865]
  Set speed (45.0 mm/s)
  Call Extruder -0.02
  MoveL (T17247) to (105.22, 121.16, 18.5) mm, rotated rx 180 ry 0 rz -180 deg; joints [1.435, 66.511, -28.949, 2.353, -37.585, -1.865]
  Set speed (150.0 mm/s)
  MoveL (T17248) to (105.22, 121.16, 20.5) mm, rotated rx 180 ry 0 rz -180 deg; joints [1.542, 66.267, -28.491, 2.517, -37.803, -1.989]
  MoveL (T17249) to (109.84, 111.88, 20.5) mm, rotated rx 180 ry 0 rz -180 deg; joints [1.542, 66.267, -28.491, 2.517, -37.803, -1.989]
  MoveL (T17250) to (109.84, 111.88, 18.5) mm, rotated rx 180 ry 0 rz -180 deg; joints [1.542, 66.267, -28.491, 2.517, -37.803, -1.989]
  Set speed (40.0 mm/s)
  Call Extruder 2.0
  MoveL (T17251) to (109.84, 111.88, 18.5) mm, rotated rx 180 ry 0 rz -180 deg; joints [1.489, 66.264, -28.485, 2.429, -37.804, -1.92]
  Set speed (31.6 mm/s)
  MoveL (T17252) to (109.84, 111.88, 18.5) mm, rotated rx 180 ry 0 rz -180 deg; joints [1.489, 66.264, -28.485, 2.429, -37.804, -1.92]
  Call Extruder 0.07441
  MoveL (T17253) to (110.95, 114.05, 18.5) mm, rotated rx 180 ry 0 rz -180 deg; joints [1.489, 66.264, -28.485, 2.429, -37.804, -1.92]
  Call Extruder 0.08223
  MoveL (T17254) to (109.04, 115.96, 18.5) mm, rotated rx 180 ry 0 rz -180 deg; joints [1.489, 66.264, -28.485, 2.429, -37.804, -1.92]
  Call Extruder 0.07057
  MoveL (T17255) to (111.36, 115.96, 18.5) mm, rotated rx 180 ry 0 rz -180 deg; joints [1.419, 66.421, -28.781, 2.322, -37.663, -1.839]
  Call Extruder 0.32359
  MoveL (T17256) to (103.84, 108.45, 18.5) mm, rotated rx 180 ry 0 rz -180 deg; joints [1.419, 66.421, -28.781, 2.322, -37.663, -1.839]
  Call Extruder 0.03385
  MoveL (T17257) to (103.84, 107.34, 18.5) mm, rotated rx 180 ry 0 rz -180 deg; joints [1.419, 66.421, -28.781, 2.322, -37.663, -1.839]
  Call Extruder 0.15054
  MoveL (T17258) to (107.34, 103.84, 18.5) mm, rotated rx 180 ry 0 rz -180 deg; joints [1.419, 66.421, -28.781, 2.322, -37.663, -1.839]
  Call Extruder 0.03385
  MoveL (T17259) to (108.45, 103.84, 18.5) mm, rotated rx 180 ry 0 rz -180 deg; joints [1.419, 66.421, -28.781, 2.322, -37.663, -1.839]
  Call Extruder 0.05679
  MoveL (T17260) to (109.77, 105.16, 18.5) mm, rotated rx 180 ry 0 rz -180 deg; joints [1.419, 66.421, -28.781, 2.322, -37.663, -1.839]
  Call Extruder 0.02614
  MoveL (T17261) to (110.63, 105.16, 18.5) mm, rotated rx 180 ry 0 rz -180 deg; joints [1.419, 66.421, -28.781, 2.322, -37.663, -1.839]
  Call Extruder 0.05679
  MoveL (T17262) to (111.94, 103.84, 18.5) mm, rotated rx 180 ry 0 rz -180 deg; joints [1.419, 66.421, -28.781, 2.322, -37.663, -1.839]
  Call Extruder 0.03385
  MoveL (T17263) to (113.06, 103.84, 18.5) mm, rotated rx 180 ry 0 rz -180 deg; joints [1.419, 66.421, -28.781, 2.322, -37.663, -1.839]
  Call Extruder 0.05679
  MoveL (T17264) to (114.37, 105.16, 18.5) mm, rotated rx 180 ry 0 rz -180 deg; joints [1.489, 66.264, -28.485, 2.429, -37.804, -1.92]
  Call Extruder 0.02614
  MoveL (T17265) to (115.23, 105.16, 18.5) mm, rotated rx 180 ry 0 rz -180 deg; joints [1.489, 66.264, -28.485, 2.429, -37.804, -1.92]
  Call Extruder 0.05679
  MoveL (T17266) to (116.55, 103.84, 18.5) mm, rotated rx 180 ry 0 rz -180 deg; joints [1.489, 66.264, -28.485, 2.429, -37.804, -1.92]
  Call Extruder 0.03385
  MoveL (T17267) to (117.66, 103.84, 18.5) mm, rotated rx 180 ry 0 rz -180 deg; joints [1.489, 66.264, -28.485, 2.429, -37.804, -1.92]
  Call Extruder 0.15054
  MoveL (T17268) to (121.16, 107.34, 18.5) mm, rotated rx 180 ry 0 rz -180 deg; joints [1.489, 66.264, -28.485, 2.429, -37.804, -1.92]
  Call Extruder 0.03385
  MoveL (T17269) to (121.16, 108.45, 18.5) mm, rotated rx 180 ry 0 rz -180 deg; joints [1.508, 66.265, -28.487, 2.461, -37.803, -1.945]
  Call Extruder 0.23679
  MoveL (T17270) to (115.66, 113.95, 18.5) mm, rotated rx 180 ry 0 rz -180 deg; joints [1.508, 66.265, -28.487, 2.461, -37.803, -1.945]
  Call Extruder 0.10426
  MoveL (T17271) to (114.1, 110.9, 18.5) mm, rotated rx 180 ry 0 rz -180 deg; joints [1.508, 66.265, -28.487, 2.461, -37.803, -1.945]
  Call Extruder 0.06615
  MoveL (T17272) to (115.64, 109.36, 18.5) mm, rotated rx 180 ry 0 rz -180 deg; joints [1.508, 66.265, -28.487, 2.461, -37.803, -1.945]
  Call Extruder 0.05076
  MoveL (T17273) to (113.97, 109.36, 18.5) mm, rotated rx 180 ry 0 rz -180 deg; joints [1.508, 66.265, -28.487, 2.461, -37.803, -1.945]
  Call Extruder 0.30958
  MoveL (T17274) to (121.16, 116.55, 18.5) mm, rotated rx 180 ry 0 rz -180 deg; joints [1.508, 66.265, -28.487, 2.461, -37.803, -1.945]
  Call Extruder 0.03385
  MoveL (T17275) to (121.16, 117.66, 18.5) mm, rotated rx 180 ry 0 rz -180 deg; joints [1.508, 66.029, -28.451, 2.472, -37.604, -1.959]
  Call Extruder 0.15054
  MoveL (T17276) to (117.66, 121.16, 18.5) mm, rotated rx 180 ry 0 rz -180 deg; joints [1.888, 67.512, -31.232, 3.188, -36.322, -2.569]
  Call Extruder 0.03385
  MoveL (T17277) to (116.55, 121.16, 18.5) mm, rotated rx 180 ry 0 rz -180 deg; joints [1.888, 67.747, -31.27, 3.173, -36.519, -2.551]
  Call Extruder 0.04278
  MoveL (T17278) to (115.56, 120.16, 18.5) mm, rotated rx 180 ry 0 rz -180 deg; joints [1.888, 67.747, -31.27, 3.173, -36.519, -2.551]
  Call Extruder 0.04595
  MoveL (T17279) to (114.05, 120.16, 18.5) mm, rotated rx 180 ry 0 rz -180 deg; joints [1.888, 67.747, -31.27, 3.173, -36.519, -2.551]
  Call Extruder 0.04278
  MoveL (T17280) to (113.06, 121.16, 18.5) mm, rotated rx 180 ry 0 rz -180 deg; joints [1.888, 67.747, -31.27, 3.173, -36.519, -2.551]
  Call Extruder 0.03385
  MoveL (T17281) to (111.94, 121.16, 18.5) mm, rotated rx 180 ry 0 rz -180 deg; joints [1.888, 67.747, -31.27, 3.173, -36.519, -2.551]
  Call Extruder 0.04278
  MoveL (T17282) to (110.95, 120.16, 18.5) mm, rotated rx 180 ry 0 rz -180 deg; joints [1.888, 67.747, -31.27, 3.173, -36.519, -2.551]
  Call Extruder 0.04595
  MoveL (T17283) to (109.44, 120.16, 18.5) mm, rotated rx 180 ry 0 rz -180 deg; joints [1.888, 67.747, -31.27, 3.173, -36.519, -2.551]
  Call Extruder 0.04278
  MoveL (T17284) to (108.45, 121.16, 18.5) mm, rotated rx 180 ry 0 rz -180 deg; joints [1.888, 67.747, -31.27, 3.173, -36.519, -2.551]
  Call Extruder 0.03385
  MoveL (T17285) to (107.34, 121.16, 18.5) mm, rotated rx 180 ry 0 rz -180 deg; joints [1.888, 67.747, -31.27, 3.173, -36.519, -2.551]
  Call Extruder 0.15054
  MoveL (T17286) to (103.84, 117.66, 18.5) mm, rotated rx 180 ry 0 rz -180 deg; joints [1.888, 67.747, -31.27, 3.173, -36.519, -2.551]
  Call Extruder 0.03385
  MoveL (T17287) to (103.84, 116.55, 18.5) mm, rotated rx 180 ry 0 rz -180 deg; joints [1.884, 68.006, -31.757, 3.184, -36.291, -2.568]
  Call Extruder 0.23899
  MoveL (T17288) to (109.39, 111, 18.5) mm, rotated rx 180 ry 0 rz -180 deg; joints [1.884, 68.006, -31.757, 3.184, -36.291, -2.568]
  Call Extruder 0.07441
  MoveL (T17289) to (108.28, 108.83, 18.5) mm, rotated rx 180 ry 0 rz -180 deg; joints [1.884, 68.006, -31.757, 3.184, -36.291, -2.568]
  Set speed (45.0 mm/s)
  Call Extruder -1.6
  MoveL (T17290) to (108.28, 108.83, 18.5) mm, rotated rx 180 ry 0 rz -180 deg; joints [1.875, 68.06, -31.858, 3.172, -36.243, -2.559]
  Set speed (120.0 mm/s)
  MoveL (T17291) to (108.28, 108.83, 18.5) mm, rotated rx 180 ry 0 rz -180 deg; joints [1.875, 68.06, -31.858, 3.172, -36.243, -2.559]
  Call Extruder -0.38
  MoveL (T17292) to (108.77, 109.78, 18.5) mm, rotated rx 180 ry 0 rz -180 deg; joints [1.875, 68.06, -31.858, 3.172, -36.243, -2.559]
  Set speed (45.0 mm/s)
  Call Extruder -0.02
  MoveL (T17293) to (108.77, 109.78, 18.5) mm, rotated rx 180 ry 0 rz -180 deg; joints [1.875, 68.06, -31.858, 3.172, -36.243, -2.559]
  Set speed (150.0 mm/s)
  MoveL (T17294) to (108.77, 109.78, 20.5) mm, rotated rx 180 ry 0 rz -180 deg; joints [1.775, 68.302, -32.313, 3.019, -36.026, -2.442]
  MoveL (T17295) to (118.71, 103.84, 20.5) mm, rotated rx 180 ry 0 rz -180 deg; joints [1.775, 68.302, -32.313, 3.019, -36.026, -2.442]
  MoveL (T17296) to (118.71, 103.84, 18.5) mm, rotated rx 180 ry 0 rz -180 deg; joints [1.775, 68.302, -32.313, 3.019, -36.026, -2.442]
  Set speed (40.0 mm/s)
  Call Extruder 2.0
  MoveL (T17297) to (118.71, 103.84, 18.5) mm, rotated rx 180 ry 0 rz -180 deg; joints [2.29, 69.793, -35.115, 4.02, -34.744, -3.305]
  Set speed (31.6 mm/s)
  MoveL (T17298) to (118.71, 103.84, 18.5) mm, rotated rx 180 ry 0 rz -180 deg; joints [2.356, 69.8, -35.129, 4.136, -34.741, -3.401]
  Call Extruder 0.07441
  MoveL (T17299) to (121.16, 103.84, 18.5) mm, rotated rx 180 ry 0 rz -180 deg; joints [2.356, 69.8, -35.129, 4.136, -34.741, -3.401]
  Call Extruder 0.13782
  MoveL (T17300) to (117.96, 107.04, 18.5) mm, rotated rx 180 ry 0 rz -180 deg; joints [3.288, 67.562, -30.924, 5.498, -36.765, -4.409]
  Call Extruder 0.05185
  MoveL (T17301) to (117.96, 108.75, 18.5) mm, rotated rx 180 ry 0 rz -180 deg; joints [3.288, 67.562, -30.924, 5.498, -36.765, -4.409]
  Call Extruder 0.13782
  MoveL (T17302) to (121.16, 111.94, 18.5) mm, rotated rx 180 ry 0 rz -180 deg; joints [3.295, 67.264, -30.364, 5.476, -37.026, -4.377]
  Call Extruder 0.03385
  MoveL (T17303) to (121.16, 113.06, 18.5) mm, rotated rx 180 ry 0 rz -180 deg; joints [3.295, 67.264, -30.364, 5.476, -37.026, -4.377]
  Call Extruder 0.16962
  MoveL (T17304) to (117.22, 116.99, 18.5) mm, rotated rx 180 ry 0 rz -180 deg; joints [2.938, 66.299, -28.551, 4.793, -37.845, -3.788]
  Call Extruder 0.01582
  MoveL (T17305) to (117.45, 117.45, 18.5) mm, rotated rx 180 ry 0 rz -180 deg; joints [2.938, 66.299, -28.551, 4.793, -37.845, -3.788]
  Call Extruder 0.15942
  MoveL (T17306) to (121.16, 121.16, 18.5) mm, rotated rx 180 ry 0 rz -180 deg; joints [2.938, 66.299, -28.551, 4.793, -37.845, -3.788]
  Call Extruder 0.07441
  MoveL (T17307) to (118.71, 121.16, 18.5) mm, rotated rx 180 ry 0 rz -180 deg; joints [2.818, 66.284, -28.524, 4.596, -37.85, -3.632]
  Set speed (45.0 mm/s)
  Call Extruder -1.6
  MoveL (T17308) to (118.71, 121.16, 18.5) mm, rotated rx 180 ry 0 rz -180 deg; joints [2.818, 66.284, -28.524, 4.596, -37.85, -3.632]
  Set speed (120.0 mm/s)
  MoveL (T17309) to (118.71, 121.16, 18.5) mm, rotated rx 180 ry 0 rz -180 deg; joints [2.818, 66.284, -28.524, 4.596, -37.85, -3.632]
  Call Extruder -0.38
  MoveL (T17310) to (119.78, 121.16, 18.5) mm, rotated rx 180 ry 0 rz -180 deg; joints [2.818, 66.284, -28.524, 4.596, -37.85, -3.632]
  Set speed (45.0 mm/s)
  Call Extruder -0.02
  MoveL (T17311) to (119.78, 121.16, 18.5) mm, rotated rx 180 ry 0 rz -180 deg; joints [1.815, 68.601, -32.874, 3.106, -35.766, -2.521]
  Set speed (150.0 mm/s)
  MoveL (T17312) to (119.78, 121.16, 20.5) mm, rotated rx 180 ry 0 rz -180 deg; joints [1.815, 68.601, -32.874, 3.106, -35.766, -2.521]
  MoveL (T17313) to (109.4, 105.47, 20.5) mm, rotated rx 180 ry 0 rz -180 deg; joints [1.815, 68.601, -32.874, 3.106, -35.766, -2.521]
  MoveL (T17314) to (109.4, 105.47, 18.7) mm, rotated rx 180 ry 0 rz -180 deg; joints [1.866, 68.745, -33.146, 3.203, -35.641, -2.604]
  Set speed (40.0 mm/s)
  Call Extruder 2.0
  MoveL (T17315) to (109.4, 105.47, 18.7) mm, rotated rx 180 ry 0 rz -180 deg; joints [1.866, 68.745, -33.146, 3.203, -35.641, -2.604]
  Set speed (31.6 mm/s)
  MoveL (T17316) to (109.4, 105.47, 18.7) mm, rotated rx 180 ry 0 rz -180 deg; joints [1.866, 68.745, -33.146, 3.203, -35.641, -2.604]
  Call Extruder 0.25145
  MoveL (T17317) to (117.65, 105.47, 18.7) mm, rotated rx 180 ry 0 rz -180 deg; joints [1.874, 68.803, -33.254, 3.221, -35.591, -2.621]
  Call Extruder 0.10939
  MoveL (T17318) to (117.65, 109.06, 18.7) mm, rotated rx 180 ry 0 rz -180 deg; joints [1.874, 68.803, -33.254, 3.221, -35.591, -2.621]
  Call Extruder 0.14732
  MoveL (T17319) to (112.81, 109.06, 18.7) mm, rotated rx 180 ry 0 rz -180 deg; joints [1.874, 68.803, -33.254, 3.221, -35.591, -2.621]
  Call Extruder 0.31102
  MoveL (T17320) to (117.47, 118.15, 18.7) mm, rotated rx 180 ry 0 rz -180 deg; joints [1.869, 69.239, -34.073, 3.243, -35.209, -2.65]
  Call Extruder 0.05209
  MoveL (T17321) to (117.47, 119.86, 18.7) mm, rotated rx 180 ry 0 rz -180 deg; joints [1.869, 69.239, -34.073, 3.243, -35.209, -2.65]
  Call Extruder 0.29244
  MoveL (T17322) to (107.87, 119.86, 18.7) mm, rotated rx 180 ry 0 rz -180 deg; joints [1.869, 69.239, -34.073, 3.243, -35.209, -2.65]
  Call Extruder 0.10939
  MoveL (T17323) to (107.87, 116.27, 18.7) mm, rotated rx 180 ry 0 rz -180 deg; joints [1.869, 69.239, -34.073, 3.243, -35.209, -2.65]
  Call Extruder 0.13869
  MoveL (T17324) to (112.42, 116.27, 18.7) mm, rotated rx 180 ry 0 rz -180 deg; joints [1.869, 69.239, -34.073, 3.243, -35.209, -2.65]
  Call Extruder 0.31084
  MoveL (T17325) to (107.78, 107.18, 18.7) mm, rotated rx 180 ry 0 rz -180 deg; joints [1.869, 69.239, -34.073, 3.243, -35.209, -2.65]
  Call Extruder 0.05206
  MoveL (T17326) to (107.78, 105.47, 18.7) mm, rotated rx 180 ry 0 rz -180 deg; joints [1.873, 68.932, -33.498, 3.228, -35.477, -2.629]
  Call Extruder 0.04735
  MoveL (T17327) to (109.34, 105.47, 18.7) mm, rotated rx 180 ry 0 rz -180 deg; joints [1.873, 68.932, -33.498, 3.228, -35.477, -2.629]
  Set speed (150.0 mm/s)
  MoveL (T17328) to (109, 105.88, 18.7) mm, rotated rx 180 ry 0 rz -180 deg; joints [1.873, 68.932, -33.498, 3.228, -35.477, -2.629]
  Set speed (31.6 mm/s)
  MoveL (T17329) to (109, 105.88, 18.7) mm, rotated rx 180 ry 0 rz -180 deg; joints [1.873, 68.932, -33.498, 3.228, -35.477, -2.629]
  Call Extruder 0.25124
  MoveL (T17330) to (117.24, 105.88, 18.7) mm, rotated rx 180 ry 0 rz -180 deg; joints [1.873, 68.698, -33.458, 3.243, -35.284, -2.648]
  Call Extruder 0.08459
  MoveL (T17331) to (117.24, 108.65, 18.7) mm, rotated rx 180 ry 0 rz -180 deg; joints [1.652, 70.823, -37.446, 3.002, -33.413, -2.506]
  Call Extruder 0.1552
  MoveL (T17332) to (112.15, 108.65, 18.7) mm, rotated rx 180 ry 0 rz -180 deg; joints [1.652, 71.056, -37.489, 2.987, -33.603, -2.488]
  Call Extruder 0.32831
  MoveL (T17333) to (117.06, 118.25, 18.7) mm, rotated rx 180 ry 0 rz -180 deg; joints [1.652, 71.056, -37.489, 2.987, -33.603, -2.488]
  Call Extruder 0.0367
  MoveL (T17334) to (117.06, 119.45, 18.7) mm, rotated rx 180 ry 0 rz -180 deg; joints [1.652, 71.056, -37.489, 2.987, -33.603, -2.488]
  Call Extruder 0.26763
  MoveL (T17335) to (108.27, 119.45, 18.7) mm, rotated rx 180 ry 0 rz -180 deg; joints [1.652, 71.056, -37.489, 2.987, -33.603, -2.488]
  Call Extruder 0.08459
  MoveL (T17336) to (108.27, 116.67, 18.7) mm, rotated rx 180 ry 0 rz -180 deg; joints [1.652, 71.056, -37.489, 2.987, -33.603, -2.488]
  Call Extruder 0.14654
  MoveL (T17337) to (113.08, 116.67, 18.7) mm, rotated rx 180 ry 0 rz -180 deg; joints [1.652, 71.056, -37.489, 2.987, -33.603, -2.488]
  Call Extruder 0.32811
  MoveL (T17338) to (108.19, 107.08, 18.7) mm, rotated rx 180 ry 0 rz -180 deg; joints [1.652, 71.056, -37.489, 2.987, -33.603, -2.488]
  Call Extruder 0.03668
  MoveL (T17339) to (108.19, 105.88, 18.7) mm, rotated rx 180 ry 0 rz -180 deg; joints [1.652, 71.056, -37.489, 2.987, -33.603, -2.488]
  Call Extruder 0.02276
  MoveL (T17340) to (108.94, 105.88, 18.7) mm, rotated rx 180 ry 0 rz -180 deg; joints [1.652, 71.056, -37.489, 2.987, -33.603, -2.488]
  Set speed (150.0 mm/s)
  MoveL (T17341) to (108.6, 106.28, 18.7) mm, rotated rx 180 ry 0 rz -180 deg; joints [1.652, 71.056, -37.489, 2.987, -33.603, -2.488]
  Set speed (25.0 mm/s)
  MoveL (T17342) to (108.6, 106.28, 18.7) mm, rotated rx 180 ry 0 rz -180 deg; joints [1.396, 71.036, -37.451, 2.522, -33.611, -2.101]
  Call Extruder 0.25102
  MoveL (T17343) to (116.84, 106.28, 18.7) mm, rotated rx 180 ry 0 rz -180 deg; joints [1.396, 71.036, -37.451, 2.522, -33.611, -2.101]
  Call Extruder 0.05979
  MoveL (T17344) to (116.84, 108.25, 18.7) mm, rotated rx 180 ry 0 rz -180 deg; joints [1.467, 70.837, -37.077, 2.638, -33.788, -2.193]
  Call Extruder 0.16307
  MoveL (T17345) to (111.48, 108.25, 18.7) mm, rotated rx 180 ry 0 rz -180 deg; joints [1.467, 70.837, -37.077, 2.638, -33.788, -2.193]
  Call Extruder 0.3456
  MoveL (T17346) to (116.65, 118.34, 18.7) mm, rotated rx 180 ry 0 rz -180 deg; joints [1.467, 70.837, -37.077, 2.638, -33.788, -2.193]
  Call Extruder 0.02131
  MoveL (T17347) to (116.65, 119.04, 18.7) mm, rotated rx 180 ry 0 rz -180 deg; joints [1.607, 70.848, -37.097, 2.89, -33.784, -2.403]
  Call Extruder 0.24283
  MoveL (T17348) to (108.68, 119.04, 18.7) mm, rotated rx 180 ry 0 rz -180 deg; joints [1.607, 70.848, -37.097, 2.89, -33.784, -2.403]
  Call Extruder 0.05979
  MoveL (T17349) to (108.68, 117.08, 18.7) mm, rotated rx 180 ry 0 rz -180 deg; joints [1.628, 70.824, -37.052, 2.927, -33.806, -2.433]
  Call Extruder 0.15438
  MoveL (T17350) to (113.75, 117.08, 18.7) mm, rotated rx 180 ry 0 rz -180 deg; joints [1.628, 70.824, -37.052, 2.927, -33.806, -2.433]
  Call Extruder 0.34538
  MoveL (T17351) to (108.6, 106.98, 18.7) mm, rotated rx 180 ry 0 rz -180 deg; joints [1.628, 70.824, -37.052, 2.927, -33.806, -2.433]
  Call Extruder 0.01947
  MoveL (T17352) to (108.6, 106.34, 18.7) mm, rotated rx 180 ry 0 rz -180 deg; joints [1.659, 70.739, -36.893, 2.976, -33.882, -2.471]
  Set speed (150.0 mm/s)
  MoveL (T17353) to (108.54, 105.89, 18.7) mm, rotated rx 180 ry 0 rz -180 deg; joints [1.659, 70.739, -36.893, 2.976, -33.882, -2.471]
  Set speed (45.0 mm/s)
  Call Extruder -1.6
  MoveL (T17354) to (108.54, 105.89, 18.7) mm, rotated rx 180 ry 0 rz -180 deg; joints [1.659, 70.739, -36.893, 2.976, -33.882, -2.471]
  Set speed (120.0 mm/s)
  MoveL (T17355) to (108.54, 105.89, 18.7) mm, rotated rx 180 ry 0 rz -180 deg; joints [1.659, 70.739, -36.893, 2.976, -33.882, -2.471]
  Call Extruder -0.38
  MoveL (T17356) to (109.66, 106.33, 18.7) mm, rotated rx 180 ry 0 rz -180 deg; joints [1.763, 71.066, -37.507, 3.187, -33.599, -2.655]
  Set speed (45.0 mm/s)
  Call Extruder -0.02
  MoveL (T17357) to (109.66, 106.33, 18.7) mm, rotated rx 180 ry 0 rz -180 deg; joints [1.763, 71.066, -37.507, 3.187, -33.599, -2.655]
  Set speed (150.0 mm/s)
  MoveL (T17358) to (109.66, 106.33, 20.7) mm, rotated rx 180 ry 0 rz -180 deg; joints [1.787, 71.068, -37.512, 3.23, -33.599, -2.692]
  MoveL (T17359) to (104.34, 103.54, 20.7) mm, rotated rx 180 ry 0 rz -180 deg; joints [1.787, 71.068, -37.512, 3.23, -33.599, -2.692]
  MoveL (T17360) to (104.34, 103.54, 18.7) mm, rotated rx 180 ry 0 rz -180 deg; joints [1.787, 71.068, -37.512, 3.23, -33.599, -2.692]
  Set speed (40.0 mm/s)
  Call Extruder 2.0
  MoveL (T17361) to (104.34, 103.54, 18.7) mm, rotated rx 180 ry 0 rz -180 deg; joints [1.787, 71.068, -37.512, 3.23, -33.599, -2.692]
  Set speed (31.6 mm/s)
  MoveL (T17362) to (104.34, 103.54, 18.7) mm, rotated rx 180 ry 0 rz -180 deg; joints [1.794, 70.439, -36.33, 3.196, -34.151, -2.646]
  Call Extruder 0.52159
  MoveL (T17363) to (121.46, 103.54, 18.7) mm, rotated rx 180 ry 0 rz -180 deg; joints [1.794, 70.439, -36.33, 3.196, -34.151, -2.646]
  Call Extruder 0.54596
  MoveL (T17364) to (121.46, 121.46, 18.7) mm, rotated rx 180 ry 0 rz -180 deg; joints [1.803, 70.379, -36.217, 3.208, -34.204, -2.654]
  Call Extruder 0.54596
  MoveL (T17365) to (103.54, 121.46, 18.7) mm, rotated rx 180 ry 0 rz -180 deg; joints [1.803, 70.379, -36.217, 3.208, -34.204, -2.654]
  Call Extruder 0.54596
  MoveL (T17366) to (103.54, 103.54, 18.7) mm, rotated rx 180 ry 0 rz -180 deg; joints [1.803, 70.379, -36.217, 3.208, -34.204, -2.654]
  Call Extruder 0.02254
  MoveL (T17367) to (104.28, 103.54, 18.7) mm, rotated rx 180 ry 0 rz -180 deg; joints [1.915, 70.08, -35.654, 3.384, -34.472, -2.791]
  Set speed (150.0 mm/s)
  MoveL (T17368) to (103.53, 103.13, 18.7) mm, rotated rx 180 ry 0 rz -180 deg; joints [1.915, 70.08, -35.654, 3.384, -34.472, -2.791]
  Set speed (31.6 mm/s)
  MoveL (T17369) to (103.53, 103.13, 18.7) mm, rotated rx 180 ry 0 rz -180 deg; joints [1.915, 70.08, -35.654, 3.384, -34.472, -2.791]
  Call Extruder 0.55858
  MoveL (T17370) to (121.87, 103.13, 18.7) mm, rotated rx 180 ry 0 rz -180 deg; joints [1.861, 69.918, -35.349, 3.277, -34.612, -2.698]
  Call Extruder 0.57077
  MoveL (T17371) to (121.87, 121.87, 18.7) mm, rotated rx 180 ry 0 rz -180 deg; joints [1.861, 69.918, -35.349, 3.277, -34.612, -2.698]
  Call Extruder 0.57077
  MoveL (T17372) to (103.13, 121.87, 18.7) mm, rotated rx 180 ry 0 rz -180 deg; joints [1.861, 69.918, -35.349, 3.277, -34.612, -2.698]
  Call Extruder 0.57077
  MoveL (T17373) to (103.13, 103.13, 18.7) mm, rotated rx 180 ry 0 rz -180 deg; joints [1.863, 69.766, -35.064, 3.269, -34.746, -2.687]
  Call Extruder 0.01036
  MoveL (T17374) to (103.47, 103.13, 18.7) mm, rotated rx 180 ry 0 rz -180 deg; joints [3.316, 66.348, -28.643, 5.412, -37.829, -4.28]
  Set speed (150.0 mm/s)
  MoveL (T17375) to (102.72, 102.81, 18.7) mm, rotated rx 180 ry 0 rz -180 deg; joints [3.316, 66.348, -28.643, 5.412, -37.829, -4.28]
  Set speed (25.0 mm/s)
  MoveL (T17376) to (102.72, 102.81, 18.7) mm, rotated rx 180 ry 0 rz -180 deg; joints [3.316, 66.348, -28.643, 5.412, -37.829, -4.28]
  Call Extruder 0.00259
  MoveL (T17377) to (102.72, 102.72, 18.7) mm, rotated rx 180 ry 0 rz -180 deg; joints [3.301, 66.985, -29.84, 5.456, -37.271, -4.347]
  Call Extruder 0.59557
  MoveL (T17378) to (122.28, 102.72, 18.7) mm, rotated rx 180 ry 0 rz -180 deg; joints [3.301, 66.985, -29.84, 5.456, -37.271, -4.347]
  Call Extruder 0.59557
  MoveL (T17379) to (122.28, 122.28, 18.7) mm, rotated rx 180 ry 0 rz -180 deg; joints [3.301, 66.985, -29.84, 5.456, -37.271, -4.347]
  Call Extruder 0.59557
  MoveL (T17380) to (102.72, 122.28, 18.7) mm, rotated rx 180 ry 0 rz -180 deg; joints [3.301, 66.985, -29.84, 5.456, -37.271, -4.347]
  Call Extruder 0.59115
  MoveL (T17381) to (102.72, 102.87, 18.7) mm, rotated rx 180 ry 0 rz -180 deg; joints [3.301, 66.985, -29.84, 5.456, -37.271, -4.347]
  Set speed (150.0 mm/s)
  MoveL (T17382) to (102.78, 102.75, 18.7) mm, rotated rx 180 ry 0 rz -180 deg; joints [3.301, 66.985, -29.84, 5.456, -37.271, -4.347]
  Set speed (45.0 mm/s)
  Call Extruder -1.6
  MoveL (T17383) to (102.78, 102.75, 18.7) mm, rotated rx 180 ry 0 rz -180 deg; joints [3.301, 66.985, -29.84, 5.456, -37.271, -4.347]
  Set speed (120.0 mm/s)
  MoveL (T17384) to (102.78, 102.75, 18.7) mm, rotated rx 180 ry 0 rz -180 deg; joints [3.301, 66.985, -29.84, 5.456, -37.271, -4.347]
  Call Extruder -0.05166
  MoveL (T17385) to (102.72, 102.72, 18.7) mm, rotated rx 180 ry 0 rz -180 deg; joints [3.301, 66.985, -29.84, 5.456, -37.271, -4.347]
  Call Extruder -0.32834
  MoveL (T17386) to (103.65, 102.72, 18.7) mm, rotated rx 180 ry 0 rz -180 deg; joints [3.301, 66.985, -29.84, 5.456, -37.271, -4.347]
  Set speed (45.0 mm/s)
  Call Extruder -0.02
  MoveL (T17387) to (103.65, 102.72, 18.7) mm, rotated rx 180 ry 0 rz -180 deg; joints [3.301, 66.985, -29.84, 5.456, -37.271, -4.347]
  Set speed (150.0 mm/s)
  MoveL (T17388) to (103.65, 102.72, 20.7) mm, rotated rx 180 ry 0 rz -180 deg; joints [3.308, 66.705, -29.314, 5.437, -37.516, -4.317]
  MoveL (T17389) to (106.29, 103.84, 20.7) mm, rotated rx 180 ry 0 rz -180 deg; joints [3.308, 66.705, -29.314, 5.437, -37.516, -4.317]
  MoveL (T17390) to (106.29, 103.84, 18.7) mm, rotated rx 180 ry 0 rz -180 deg; joints [3.308, 66.705, -29.314, 5.437, -37.516, -4.317]
  Set speed (40.0 mm/s)
  Call Extruder 2.0
  MoveL (T17391) to (106.29, 103.84, 18.7) mm, rotated rx 180 ry 0 rz -180 deg; joints [3.308, 66.705, -29.314, 5.437, -37.516, -4.317]
  Set speed (31.6 mm/s)
  MoveL (T17392) to (106.29, 103.84, 18.7) mm, rotated rx 180 ry 0 rz -180 deg; joints [3.308, 66.705, -29.314, 5.437, -37.516, -4.317]
  Call Extruder 0.07441
  MoveL (T17393) to (103.84, 103.84, 18.7) mm, rotated rx 180 ry 0 rz -180 deg; joints [1.407, 66.052, -28.494, 2.308, -37.58, -1.829]
  Call Extruder 0.16673
  MoveL (T17394) to (107.71, 107.71, 18.7) mm, rotated rx 180 ry 0 rz -180 deg; joints [1.407, 66.264, -28.527, 2.299, -37.76, -1.818]
  Call Extruder 0.00815
  MoveL (T17395) to (107.84, 107.95, 18.7) mm, rotated rx 180 ry 0 rz -180 deg; joints [1.407, 66.264, -28.527, 2.299, -37.76, -1.818]
  Call Extruder 0.17197
  MoveL (T17396) to (103.84, 111.94, 18.7) mm, rotated rx 180 ry 0 rz -180 deg; joints [1.407, 66.264, -28.527, 2.299, -37.76, -1.818]
  Call Extruder 0.03385
  MoveL (T17397) to (103.84, 113.06, 18.7) mm, rotated rx 180 ry 0 rz -180 deg; joints [1.407, 66.264, -28.527, 2.299, -37.76, -1.818]
  Call Extruder 0.16015
  MoveL (T17398) to (107.56, 116.77, 18.7) mm, rotated rx 180 ry 0 rz -180 deg; joints [1.407, 66.264, -28.527, 2.299, -37.76, -1.818]
  Call Extruder 0.02027
  MoveL (T17399) to (107.56, 117.44, 18.7) mm, rotated rx 180 ry 0 rz -180 deg; joints [1.407, 66.264, -28.527, 2.299, -37.76, -1.818]
  Call Extruder 0.16015
  MoveL (T17400) to (103.84, 121.16, 18.7) mm, rotated rx 180 ry 0 rz -180 deg; joints [1.407, 66.264, -28.527, 2.299, -37.76, -1.818]
  Call Extruder 0.07441
  MoveL (T17401) to (106.29, 121.16, 18.7) mm, rotated rx 180 ry 0 rz -180 deg; joints [1.407, 66.264, -28.527, 2.299, -37.76, -1.818]
  Set speed (45.0 mm/s)
  Call Extruder -1.6
  MoveL (T17402) to (106.29, 121.16, 18.7) mm, rotated rx 180 ry 0 rz -180 deg; joints [1.407, 66.264, -28.527, 2.299, -37.76, -1.818]
  Set speed (120.0 mm/s)
  MoveL (T17403) to (106.29, 121.16, 18.7) mm, rotated rx 180 ry 0 rz -180 deg; joints [1.407, 66.264, -28.527, 2.299, -37.76, -1.818]
  Call Extruder -0.38
  MoveL (T17404) to (105.22, 121.16, 18.7) mm, rotated rx 180 ry 0 rz -180 deg; joints [1.363, 71.106, -37.621, 2.47, -33.509, -2.06]
  Set speed (45.0 mm/s)
  Call Extruder -0.02
  MoveL (T17405) to (105.22, 121.16, 18.7) mm, rotated rx 180 ry 0 rz -180 deg; joints [1.363, 71.106, -37.621, 2.47, -33.509, -2.06]
  Set speed (150.0 mm/s)
  MoveL (T17406) to (105.22, 121.16, 20.7) mm, rotated rx 180 ry 0 rz -180 deg; joints [1.363, 71.106, -37.621, 2.47, -33.509, -2.06]
  MoveL (T17407) to (109.84, 111.88, 20.7) mm, rotated rx 180 ry 0 rz -180 deg; joints [1.363, 71.106, -37.621, 2.47, -33.509, -2.06]
  MoveL (T17408) to (109.84, 111.88, 18.7) mm, rotated rx 180 ry 0 rz -180 deg; joints [3.241, 71.333, -38.048, 5.892, -33.424, -4.923]
  Set speed (40.0 mm/s)
  Call Extruder 2.0
  MoveL (T17409) to (109.84, 111.88, 18.7) mm, rotated rx 180 ry 0 rz -180 deg; joints [3.241, 71.333, -38.048, 5.892, -33.424, -4.923]
  Set speed (31.6 mm/s)
  MoveL (T17410) to (109.84, 111.88, 18.7) mm, rotated rx 180 ry 0 rz -180 deg; joints [3.241, 71.333, -38.048, 5.892, -33.424, -4.923]
  Call Extruder 0.07441
  MoveL (T17411) to (110.95, 114.05, 18.7) mm, rotated rx 180 ry 0 rz -180 deg; joints [3.241, 71.333, -38.048, 5.892, -33.424, -4.923]
  Call Extruder 0.08223
  MoveL (T17412) to (109.04, 115.96, 18.7) mm, rotated rx 180 ry 0 rz -180 deg; joints [3.351, 66.25, -28.5, 5.463, -37.876, -4.317]
  Call Extruder 0.07057
  MoveL (T17413) to (111.36, 115.96, 18.7) mm, rotated rx 180 ry 0 rz -180 deg; joints [3.351, 66.25, -28.5, 5.463, -37.876, -4.317]
  Call Extruder 0.32359
  MoveL (T17414) to (103.84, 108.45, 18.7) mm, rotated rx 180 ry 0 rz -180 deg; joints [3.351, 66.25, -28.5, 5.463, -37.876, -4.317]
  Call Extruder 0.03385
  MoveL (T17415) to (103.84, 107.34, 18.7) mm, rotated rx 180 ry 0 rz -180 deg; joints [1.409, 66.059, -28.142, 2.293, -37.94, -1.809]
  Call Extruder 0.15054
  MoveL (T17416) to (107.34, 103.84, 18.7) mm, rotated rx 180 ry 0 rz -180 deg; joints [1.409, 66.059, -28.142, 2.293, -37.94, -1.809]
  Call Extruder 0.03385
  MoveL (T17417) to (108.45, 103.84, 18.7) mm, rotated rx 180 ry 0 rz -180 deg; joints [1.409, 66.059, -28.142, 2.293, -37.94, -1.809]
  Call Extruder 0.05679
  MoveL (T17418) to (109.77, 105.16, 18.7) mm, rotated rx 180 ry 0 rz -180 deg; joints [1.409, 66.059, -28.142, 2.293, -37.94, -1.809]
  Call Extruder 0.02614
  MoveL (T17419) to (110.63, 105.16, 18.7) mm, rotated rx 180 ry 0 rz -180 deg; joints [1.407, 66.249, -28.498, 2.298, -37.773, -1.817]
  Call Extruder 0.05679
  MoveL (T17420) to (111.94, 103.84, 18.7) mm, rotated rx 180 ry 0 rz -180 deg; joints [1.407, 66.249, -28.498, 2.298, -37.773, -1.817]
  Call Extruder 0.03385
  MoveL (T17421) to (113.06, 103.84, 18.7) mm, rotated rx 180 ry 0 rz -180 deg; joints [1.365, 66.055, -28.133, 2.221, -37.942, -1.752]
  Call Extruder 0.05679
  MoveL (T17422) to (114.37, 105.16, 18.7) mm, rotated rx 180 ry 0 rz -180 deg; joints [1.365, 66.055, -28.133, 2.221, -37.942, -1.752]
  Call Extruder 0.02614
  MoveL (T17423) to (115.23, 105.16, 18.7) mm, rotated rx 180 ry 0 rz -180 deg; joints [1.365, 66.055, -28.133, 2.221, -37.942, -1.752]
  Call Extruder 0.05679
  MoveL (T17424) to (116.55, 103.84, 18.7) mm, rotated rx 180 ry 0 rz -180 deg; joints [1.365, 66.055, -28.133, 2.221, -37.942, -1.752]
  Call Extruder 0.03385
  MoveL (T17425) to (117.66, 103.84, 18.7) mm, rotated rx 180 ry 0 rz -180 deg; joints [1.365, 66.055, -28.133, 2.221, -37.942, -1.752]
  Call Extruder 0.15054
  MoveL (T17426) to (121.16, 107.34, 18.7) mm, rotated rx 180 ry 0 rz -180 deg; joints [1.365, 66.055, -28.133, 2.221, -37.942, -1.752]
  Call Extruder 0.03385
  MoveL (T17427) to (121.16, 108.45, 18.7) mm, rotated rx 180 ry 0 rz -180 deg; joints [1.319, 71.231, -37.856, 2.398, -33.397, -2.002]
  Call Extruder 0.23679
  MoveL (T17428) to (115.66, 113.95, 18.7) mm, rotated rx 180 ry 0 rz -180 deg; joints [1.319, 71.231, -37.856, 2.398, -33.397, -2.002]
  Call Extruder 0.10426
  MoveL (T17429) to (114.1, 110.9, 18.7) mm, rotated rx 180 ry 0 rz -180 deg; joints [1.319, 71.231, -37.856, 2.398, -33.397, -2.002]
  Call Extruder 0.06615
  MoveL (T17430) to (115.64, 109.36, 18.7) mm, rotated rx 180 ry 0 rz -180 deg; joints [3.282, 71.469, -38.305, 5.983, -33.308, -5.006]
  Call Extruder 0.05076
  MoveL (T17431) to (113.97, 109.36, 18.7) mm, rotated rx 180 ry 0 rz -180 deg; joints [3.282, 71.469, -38.305, 5.983, -33.308, -5.006]
  Call Extruder 0.30958
  MoveL (T17432) to (121.16, 116.55, 18.7) mm, rotated rx 180 ry 0 rz -180 deg; joints [3.282, 71.469, -38.305, 5.983, -33.308, -5.006]
  Call Extruder 0.03385
  MoveL (T17433) to (121.16, 117.66, 18.7) mm, rotated rx 180 ry 0 rz -180 deg; joints [3.282, 71.469, -38.305, 5.983, -33.308, -5.006]
  Call Extruder 0.15054
  MoveL (T17434) to (117.66, 121.16, 18.7) mm, rotated rx 180 ry 0 rz -180 deg; joints [3.398, 66.152, -28.316, 5.529, -37.966, -4.364]
  Call Extruder 0.03385
  MoveL (T17435) to (116.55, 121.16, 18.7) mm, rotated rx 180 ry 0 rz -180 deg; joints [3.398, 66.152, -28.316, 5.529, -37.966, -4.364]
  Call Extruder 0.04278
  MoveL (T17436) to (115.56, 120.16, 18.7) mm, rotated rx 180 ry 0 rz -180 deg; joints [3.398, 66.152, -28.316, 5.529, -37.966, -4.364]
  Call Extruder 0.04595
  MoveL (T17437) to (114.05, 120.16, 18.7) mm, rotated rx 180 ry 0 rz -180 deg; joints [3.398, 66.152, -28.316, 5.529, -37.966, -4.364]
  Call Extruder 0.04278
  MoveL (T17438) to (113.06, 121.16, 18.7) mm, rotated rx 180 ry 0 rz -180 deg; joints [3.398, 66.152, -28.316, 5.529, -37.966, -4.364]
  Call Extruder 0.03385
  MoveL (T17439) to (111.94, 121.16, 18.7) mm, rotated rx 180 ry 0 rz -180 deg; joints [1.366, 65.953, -27.942, 2.218, -38.032, -1.747]
  Call Extruder 0.04278
  MoveL (T17440) to (110.95, 120.16, 18.7) mm, rotated rx 180 ry 0 rz -180 deg; joints [1.366, 65.953, -27.942, 2.218, -38.032, -1.747]
  Call Extruder 0.04595
  MoveL (T17441) to (109.44, 120.16, 18.7) mm, rotated rx 180 ry 0 rz -180 deg; joints [1.366, 65.953, -27.942, 2.218, -38.032, -1.747]
  Call Extruder 0.04278
  MoveL (T17442) to (108.45, 121.16, 18.7) mm, rotated rx 180 ry 0 rz -180 deg; joints [1.365, 66.039, -28.105, 2.22, -37.956, -1.751]
  Call Extruder 0.03385
  MoveL (T17443) to (107.34, 121.16, 18.7) mm, rotated rx 180 ry 0 rz -180 deg; joints [1.365, 66.039, -28.105, 2.22, -37.956, -1.751]
  Call Extruder 0.15054
  MoveL (T17444) to (103.84, 117.66, 18.7) mm, rotated rx 180 ry 0 rz -180 deg; joints [1.365, 66.039, -28.105, 2.22, -37.956, -1.751]
  Call Extruder 0.03385
  MoveL (T17445) to (103.84, 116.55, 18.7) mm, rotated rx 180 ry 0 rz -180 deg; joints [1.365, 66.039, -28.105, 2.22, -37.956, -1.751]
  Call Extruder 0.23899
  MoveL (T17446) to (109.39, 111, 18.7) mm, rotated rx 180 ry 0 rz -180 deg; joints [1.332, 65.847, -27.744, 2.159, -38.123, -1.698]
  Call Extruder 0.07441
  MoveL (T17447) to (108.28, 108.83, 18.7) mm, rotated rx 180 ry 0 rz -180 deg; joints [1.332, 65.847, -27.744, 2.159, -38.123, -1.698]
  Set speed (45.0 mm/s)
  Call Extruder -1.6
  MoveL (T17448) to (108.28, 108.83, 18.7) mm, rotated rx 180 ry 0 rz -180 deg; joints [1.332, 65.847, -27.744, 2.159, -38.123, -1.698]
  Set speed (120.0 mm/s)
  MoveL (T17449) to (108.28, 108.83, 18.7) mm, rotated rx 180 ry 0 rz -180 deg; joints [1.332, 65.847, -27.744, 2.159, -38.123, -1.698]
  Call Extruder -0.38
  MoveL (T17450) to (108.77, 109.78, 18.7) mm, rotated rx 180 ry 0 rz -180 deg; joints [1.332, 65.847, -27.744, 2.159, -38.123, -1.698]
  Set speed (45.0 mm/s)
  Call Extruder -0.02
  MoveL (T17451) to (108.77, 109.78, 18.7) mm, rotated rx 180 ry 0 rz -180 deg; joints [1.323, 65.847, -27.743, 2.144, -38.123, -1.687]
  Set speed (150.0 mm/s)
  MoveL (T17452) to (108.77, 109.78, 20.7) mm, rotated rx 180 ry 0 rz -180 deg; joints [1.276, 71.356, -38.093, 2.325, -33.285, -1.944]
  MoveL (T17453) to (118.71, 103.84, 20.7) mm, rotated rx 180 ry 0 rz -180 deg; joints [1.276, 71.356, -38.093, 2.325, -33.285, -1.944]
  MoveL (T17454) to (118.71, 103.84, 18.7) mm, rotated rx 180 ry 0 rz -180 deg; joints [1.276, 71.356, -38.093, 2.325, -33.285, -1.944]
  Set speed (40.0 mm/s)
  Call Extruder 2.0
  MoveL (T17455) to (118.71, 103.84, 18.7) mm, rotated rx 180 ry 0 rz -180 deg; joints [1.276, 71.356, -38.093, 2.325, -33.285, -1.944]
  Set speed (31.6 mm/s)
  MoveL (T17456) to (118.71, 103.84, 18.7) mm, rotated rx 180 ry 0 rz -180 deg; joints [3.322, 71.607, -38.563, 6.076, -33.191, -5.09]
  Call Extruder 0.07441
  MoveL (T17457) to (121.16, 103.84, 18.7) mm, rotated rx 180 ry 0 rz -180 deg; joints [3.322, 71.607, -38.563, 6.076, -33.191, -5.09]
  Call Extruder 0.13782
  MoveL (T17458) to (117.96, 107.04, 18.7) mm, rotated rx 180 ry 0 rz -180 deg; joints [3.322, 71.607, -38.563, 6.076, -33.191, -5.09]
  Call Extruder 0.05185
  MoveL (T17459) to (117.96, 108.75, 18.7) mm, rotated rx 180 ry 0 rz -180 deg; joints [3.322, 71.607, -38.563, 6.076, -33.191, -5.09]
  Call Extruder 0.13782
  MoveL (T17460) to (121.16, 111.94, 18.7) mm, rotated rx 180 ry 0 rz -180 deg; joints [3.445, 66.054, -28.132, 5.593, -38.055, -4.41]
  Call Extruder 0.03385
  MoveL (T17461) to (121.16, 113.06, 18.7) mm, rotated rx 180 ry 0 rz -180 deg; joints [3.445, 66.054, -28.132, 5.593, -38.055, -4.41]
  Call Extruder 0.16962
  MoveL (T17462) to (117.22, 116.99, 18.7) mm, rotated rx 180 ry 0 rz -180 deg; joints [3.445, 66.054, -28.132, 5.593, -38.055, -4.41]
  Call Extruder 0.01582
  MoveL (T17463) to (117.45, 117.45, 18.7) mm, rotated rx 180 ry 0 rz -180 deg; joints [1.339, 65.848, -27.744, 2.169, -38.123, -1.707]
  Call Extruder 0.15942
  MoveL (T17464) to (121.16, 121.16, 18.7) mm, rotated rx 180 ry 0 rz -180 deg; joints [1.339, 65.848, -27.744, 2.169, -38.123, -1.707]
  Call Extruder 0.07441
  MoveL (T17465) to (118.71, 121.16, 18.7) mm, rotated rx 180 ry 0 rz -180 deg; joints [1.339, 65.848, -27.744, 2.169, -38.123, -1.707]
  Set speed (45.0 mm/s)
  Call Extruder -1.6
  MoveL (T17466) to (118.71, 121.16, 18.7) mm, rotated rx 180 ry 0 rz -180 deg; joints [1.339, 65.848, -27.744, 2.169, -38.123, -1.707]
  Set speed (120.0 mm/s)
  MoveL (T17467) to (118.71, 121.16, 18.7) mm, rotated rx 180 ry 0 rz -180 deg; joints [1.326, 65.862, -27.772, 2.148, -38.11, -1.691]
  Call Extruder -0.38
  MoveL (T17468) to (119.78, 121.16, 18.7) mm, rotated rx 180 ry 0 rz -180 deg; joints [1.326, 65.862, -27.772, 2.148, -38.11, -1.691]
  Set speed (45.0 mm/s)
  Call Extruder -0.02
  MoveL (T17469) to (119.78, 121.16, 18.7) mm, rotated rx 180 ry 0 rz -180 deg; joints [1.326, 65.862, -27.772, 2.148, -38.11, -1.691]
  Set speed (150.0 mm/s)
  MoveL (T17470) to (119.78, 121.16, 20.7) mm, rotated rx 180 ry 0 rz -180 deg; joints [1.326, 65.862, -27.772, 2.148, -38.11, -1.691]
  MoveL (T17471) to (109.4, 105.47, 20.7) mm, rotated rx 180 ry 0 rz -180 deg; joints [1.326, 65.862, -27.772, 2.148, -38.11, -1.691]
  MoveL (T17472) to (109.4, 105.47, 18.9) mm, rotated rx 180 ry 0 rz -180 deg; joints [1.326, 65.862, -27.772, 2.148, -38.11, -1.691]
  Set speed (40.0 mm/s)
  Call Extruder 2.0
  MoveL (T17473) to (109.4, 105.47, 18.9) mm, rotated rx 180 ry 0 rz -180 deg; joints [1.326, 65.862, -27.772, 2.148, -38.11, -1.691]
  Call Extruder 0.25145
  MoveL (T17474) to (117.65, 105.47, 18.9) mm, rotated rx 180 ry 0 rz -180 deg; joints [1.326, 65.862, -27.772, 2.148, -38.11, -1.691]
  Call Extruder 0.10939
  MoveL (T17475) to (117.65, 109.06, 18.9) mm, rotated rx 180 ry 0 rz -180 deg; joints [1.326, 65.862, -27.772, 2.148, -38.11, -1.691]
  Call Extruder 0.14732
  MoveL (T17476) to (112.81, 109.06, 18.9) mm, rotated rx 180 ry 0 rz -180 deg; joints [1.323, 65.847, -27.743, 2.144, -38.123, -1.687]
  Call Extruder 0.31102
  MoveL (T17477) to (117.47, 118.15, 18.9) mm, rotated rx 180 ry 0 rz -180 deg; joints [1.323, 65.847, -27.743, 2.144, -38.123, -1.687]
  Call Extruder 0.05209
  MoveL (T17478) to (117.47, 119.86, 18.9) mm, rotated rx 180 ry 0 rz -180 deg; joints [1.321, 66.082, -28.184, 2.15, -37.917, -1.696]
  Call Extruder 0.29244
  MoveL (T17479) to (107.87, 119.86, 18.9) mm, rotated rx 180 ry 0 rz -180 deg; joints [1.321, 66.082, -28.184, 2.15, -37.917, -1.696]
  Call Extruder 0.10939
  MoveL (T17480) to (107.87, 116.27, 18.9) mm, rotated rx 180 ry 0 rz -180 deg; joints [1.321, 66.082, -28.184, 2.15, -37.917, -1.696]
  Call Extruder 0.13869
  MoveL (T17481) to (112.42, 116.27, 18.9) mm, rotated rx 180 ry 0 rz -180 deg; joints [1.321, 66.082, -28.184, 2.15, -37.917, -1.696]
  Call Extruder 0.31084
  MoveL (T17482) to (107.78, 107.18, 18.9) mm, rotated rx 180 ry 0 rz -180 deg; joints [1.321, 66.082, -28.184, 2.15, -37.917, -1.696]
  Call Extruder 0.05206
  MoveL (T17483) to (107.78, 105.47, 18.9) mm, rotated rx 180 ry 0 rz -180 deg; joints [1.321, 66.082, -28.184, 2.15, -37.917, -1.696]
  Call Extruder 0.04735
  MoveL (T17484) to (109.34, 105.47, 18.9) mm, rotated rx 180 ry 0 rz -180 deg; joints [1.321, 66.082, -28.184, 2.15, -37.917, -1.696]
  Set speed (150.0 mm/s)
  MoveL (T17485) to (109, 105.88, 18.9) mm, rotated rx 180 ry 0 rz -180 deg; joints [1.707, 65.92, -28.288, 2.793, -37.665, -2.212]
  Set speed (40.0 mm/s)
  MoveL (T17486) to (109, 105.88, 18.9) mm, rotated rx 180 ry 0 rz -180 deg; joints [1.707, 65.92, -28.288, 2.793, -37.665, -2.212]
  Call Extruder 0.25124
  MoveL (T17487) to (117.24, 105.88, 18.9) mm, rotated rx 180 ry 0 rz -180 deg; joints [1.707, 66.156, -28.324, 2.781, -37.865, -2.196]
  Call Extruder 0.08459
  MoveL (T17488) to (117.24, 108.65, 18.9) mm, rotated rx 180 ry 0 rz -180 deg; joints [1.707, 66.156, -28.324, 2.781, -37.865, -2.196]
  Call Extruder 0.1552
  MoveL (T17489) to (112.15, 108.65, 18.9) mm, rotated rx 180 ry 0 rz -180 deg; joints [1.707, 66.156, -28.324, 2.781, -37.865, -2.196]
  Call Extruder 0.32831
  MoveL (T17490) to (117.06, 118.25, 18.9) mm, rotated rx 180 ry 0 rz -180 deg; joints [1.707, 66.156, -28.324, 2.781, -37.865, -2.196]
  Call Extruder 0.0367
  MoveL (T17491) to (117.06, 119.45, 18.9) mm, rotated rx 180 ry 0 rz -180 deg; joints [1.707, 66.156, -28.324, 2.781, -37.865, -2.196]
  Call Extruder 0.26763
  MoveL (T17492) to (108.27, 119.45, 18.9) mm, rotated rx 180 ry 0 rz -180 deg; joints [1.707, 66.156, -28.324, 2.781, -37.865, -2.196]
  Call Extruder 0.08459
  MoveL (T17493) to (108.27, 116.67, 18.9) mm, rotated rx 180 ry 0 rz -180 deg; joints [1.707, 66.156, -28.324, 2.781, -37.865, -2.196]
  Call Extruder 0.14654
  MoveL (T17494) to (113.08, 116.67, 18.9) mm, rotated rx 180 ry 0 rz -180 deg; joints [1.707, 66.156, -28.324, 2.781, -37.865, -2.196]
  Call Extruder 0.32811
  MoveL (T17495) to (108.19, 107.08, 18.9) mm, rotated rx 180 ry 0 rz -180 deg; joints [1.707, 66.156, -28.324, 2.781, -37.865, -2.196]
  Call Extruder 0.03668
  MoveL (T17496) to (108.19, 105.88, 18.9) mm, rotated rx 180 ry 0 rz -180 deg; joints [1.442, 66.139, -28.292, 2.349, -37.871, -1.855]
  Call Extruder 0.02276
  MoveL (T17497) to (108.94, 105.88, 18.9) mm, rotated rx 180 ry 0 rz -180 deg; joints [1.442, 66.139, -28.292, 2.349, -37.871, -1.855]
  Set speed (150.0 mm/s)
  MoveL (T17498) to (108.6, 106.28, 18.9) mm, rotated rx 180 ry 0 rz -180 deg; joints [1.657, 66.154, -28.32, 2.7, -37.865, -2.133]
  Set speed (25.0 mm/s)
  MoveL (T17499) to (108.6, 106.28, 18.9) mm, rotated rx 180 ry 0 rz -180 deg; joints [1.657, 66.154, -28.32, 2.7, -37.865, -2.133]
  Call Extruder 0.25102
  MoveL (T17500) to (116.84, 106.28, 18.9) mm, rotated rx 180 ry 0 rz -180 deg; joints [1.679, 66.177, -28.363, 2.737, -37.846, -2.162]
  Call Extruder 0.05979
  MoveL (T17501) to (116.84, 108.25, 18.9) mm, rotated rx 180 ry 0 rz -180 deg; joints [1.679, 66.177, -28.363, 2.737, -37.846, -2.162]
  Call Extruder 0.16307
  MoveL (T17502) to (111.48, 108.25, 18.9) mm, rotated rx 180 ry 0 rz -180 deg; joints [1.679, 66.177, -28.363, 2.737, -37.846, -2.162]
  Call Extruder 0.3456
  MoveL (T17503) to (116.65, 118.34, 18.9) mm, rotated rx 180 ry 0 rz -180 deg; joints [1.679, 66.177, -28.363, 2.737, -37.846, -2.162]
  Call Extruder 0.02131
  MoveL (T17504) to (116.65, 119.04, 18.9) mm, rotated rx 180 ry 0 rz -180 deg; joints [1.679, 66.177, -28.363, 2.737, -37.846, -2.162]
  Call Extruder 0.24283
  MoveL (T17505) to (108.68, 119.04, 18.9) mm, rotated rx 180 ry 0 rz -180 deg; joints [1.743, 66.339, -28.666, 2.85, -37.707, -2.256]
  Call Extruder 0.05979
  MoveL (T17506) to (108.68, 117.08, 18.9) mm, rotated rx 180 ry 0 rz -180 deg; joints [1.743, 66.339, -28.666, 2.85, -37.707, -2.256]
  Call Extruder 0.15438
  MoveL (T17507) to (113.75, 117.08, 18.9) mm, rotated rx 180 ry 0 rz -180 deg; joints [1.821, 66.165, -28.34, 2.967, -37.862, -2.343]
  Call Extruder 0.34538
  MoveL (T17508) to (108.6, 106.98, 18.9) mm, rotated rx 180 ry 0 rz -180 deg; joints [1.821, 66.165, -28.34, 2.967, -37.862, -2.343]
  Call Extruder 0.01947
  MoveL (T17509) to (108.6, 106.34, 18.9) mm, rotated rx 180 ry 0 rz -180 deg; joints [1.821, 66.165, -28.34, 2.967, -37.862, -2.343]
  Set speed (150.0 mm/s)
  MoveL (T17510) to (108.54, 105.89, 18.9) mm, rotated rx 180 ry 0 rz -180 deg; joints [1.821, 66.165, -28.34, 2.967, -37.862, -2.343]
  Set speed (45.0 mm/s)
  Call Extruder -1.6
  MoveL (T17511) to (108.54, 105.89, 18.9) mm, rotated rx 180 ry 0 rz -180 deg; joints [1.821, 66.165, -28.34, 2.967, -37.862, -2.343]
  Set speed (120.0 mm/s)
  MoveL (T17512) to (108.54, 105.89, 18.9) mm, rotated rx 180 ry 0 rz -180 deg; joints [1.941, 66.174, -28.357, 3.164, -37.859, -2.499]
  Call Extruder -0.38
  MoveL (T17513) to (109.66, 106.33, 18.9) mm, rotated rx 180 ry 0 rz -180 deg; joints [1.941, 66.174, -28.357, 3.164, -37.859, -2.499]
  Set speed (45.0 mm/s)
  Call Extruder -0.02
  MoveL (T17514) to (109.66, 106.33, 18.9) mm, rotated rx 180 ry 0 rz -180 deg; joints [3.239, 69.825, -35.215, 5.689, -34.742, -4.68]
  Set speed (150.0 mm/s)
  MoveL (T17515) to (109.66, 106.33, 20.9) mm, rotated rx 180 ry 0 rz -180 deg; joints [3.239, 69.825, -35.215, 5.689, -34.742, -4.68]
  MoveL (T17516) to (104.34, 103.54, 20.9) mm, rotated rx 180 ry 0 rz -180 deg; joints [3.239, 69.825, -35.215, 5.689, -34.742, -4.68]
  MoveL (T17517) to (104.34, 103.54, 18.9) mm, rotated rx 180 ry 0 rz -180 deg; joints [3.232, 70.156, -35.837, 5.719, -34.452, -4.721]
  Set speed (40.0 mm/s)
  Call Extruder 2.0
  MoveL (T17518) to (104.34, 103.54, 18.9) mm, rotated rx 180 ry 0 rz -180 deg; joints [3.232, 70.156, -35.837, 5.719, -34.452, -4.721]
  Call Extruder 0.52159
  MoveL (T17519) to (121.46, 103.54, 18.9) mm, rotated rx 180 ry 0 rz -180 deg; joints [2.845, 71.173, -37.748, 5.155, -33.532, -4.301]
  Call Extruder 0.54596
  MoveL (T17520) to (121.46, 121.46, 18.9) mm, rotated rx 180 ry 0 rz -180 deg; joints [2.845, 71.173, -37.748, 5.155, -33.532, -4.301]
  Call Extruder 0.54596
  MoveL (T17521) to (103.54, 121.46, 18.9) mm, rotated rx 180 ry 0 rz -180 deg; joints [2.845, 71.173, -37.748, 5.155, -33.532, -4.301]
  Call Extruder 0.54596
  MoveL (T17522) to (103.54, 103.54, 18.9) mm, rotated rx 180 ry 0 rz -180 deg; joints [3.211, 71.231, -37.857, 5.824, -33.51, -4.861]
  Call Extruder 0.02254
  MoveL (T17523) to (104.28, 103.54, 18.9) mm, rotated rx 180 ry 0 rz -180 deg; joints [3.211, 71.231, -37.857, 5.824, -33.51, -4.861]
  Set speed (150.0 mm/s)
  MoveL (T17524) to (103.53, 103.13, 18.9) mm, rotated rx 180 ry 0 rz -180 deg; joints [3.211, 71.231, -37.857, 5.824, -33.51, -4.861]
  Set speed (40.0 mm/s)
  MoveL (T17525) to (103.53, 103.13, 18.9) mm, rotated rx 180 ry 0 rz -180 deg; joints [1.893, 67.3, -30.472, 3.156, -36.87, -2.526]
  Call Extruder 0.55858
  MoveL (T17526) to (121.87, 103.13, 18.9) mm, rotated rx 180 ry 0 rz -180 deg; joints [1.893, 67.3, -30.472, 3.156, -36.87, -2.526]
  Call Extruder 0.57077
  MoveL (T17527) to (121.87, 121.87, 18.9) mm, rotated rx 180 ry 0 rz -180 deg; joints [1.893, 67.3, -30.472, 3.156, -36.87, -2.526]
  Call Extruder 0.57077
  MoveL (T17528) to (103.13, 121.87, 18.9) mm, rotated rx 180 ry 0 rz -180 deg; joints [1.893, 67.3, -30.472, 3.156, -36.87, -2.526]
  Call Extruder 0.57077
  MoveL (T17529) to (103.13, 103.13, 18.9) mm, rotated rx 180 ry 0 rz -180 deg; joints [1.895, 67.163, -30.215, 3.15, -36.99, -2.517]
  Call Extruder 0.01036
  MoveL (T17530) to (103.47, 103.13, 18.9) mm, rotated rx 180 ry 0 rz -180 deg; joints [1.895, 67.163, -30.215, 3.15, -36.99, -2.517]
  Set speed (150.0 mm/s)
  MoveL (T17531) to (102.72, 102.81, 18.9) mm, rotated rx 180 ry 0 rz -180 deg; joints [2.319, 66.207, -28.42, 3.782, -37.848, -2.988]
  Set speed (25.0 mm/s)
  MoveL (T17532) to (102.72, 102.81, 18.9) mm, rotated rx 180 ry 0 rz -180 deg; joints [2.319, 66.207, -28.42, 3.782, -37.848, -2.988]
  Call Extruder 0.00259
  MoveL (T17533) to (102.72, 102.72, 18.9) mm, rotated rx 180 ry 0 rz -180 deg; joints [2.319, 66.207, -28.42, 3.782, -37.848, -2.988]
  Call Extruder 0.59557
  MoveL (T17534) to (122.28, 102.72, 18.9) mm, rotated rx 180 ry 0 rz -180 deg; joints [2.319, 66.207, -28.42, 3.782, -37.848, -2.988]
  Call Extruder 0.59557
  MoveL (T17535) to (122.28, 122.28, 18.9) mm, rotated rx 180 ry 0 rz -180 deg; joints [2.44, 66.219, -28.442, 3.979, -37.844, -3.144]
  Call Extruder 0.59557
  MoveL (T17536) to (102.72, 122.28, 18.9) mm, rotated rx 180 ry 0 rz -180 deg; joints [2.44, 66.219, -28.442, 3.979, -37.844, -3.144]
  Call Extruder 0.59115
  MoveL (T17537) to (102.72, 102.87, 18.9) mm, rotated rx 180 ry 0 rz -180 deg; joints [2.44, 66.219, -28.442, 3.979, -37.844, -3.144]
  Set speed (150.0 mm/s)
  MoveL (T17538) to (102.78, 102.75, 18.9) mm, rotated rx 180 ry 0 rz -180 deg; joints [3.266, 68.499, -32.724, 5.576, -35.904, -4.521]
  Set speed (45.0 mm/s)
  Call Extruder -1.6
  MoveL (T17539) to (102.78, 102.75, 18.9) mm, rotated rx 180 ry 0 rz -180 deg; joints [3.266, 68.499, -32.724, 5.576, -35.904, -4.521]
  Set speed (120.0 mm/s)
  MoveL (T17540) to (102.78, 102.75, 18.9) mm, rotated rx 180 ry 0 rz -180 deg; joints [3.266, 68.499, -32.724, 5.576, -35.904, -4.521]
  Call Extruder -0.05166
  MoveL (T17541) to (102.72, 102.72, 18.9) mm, rotated rx 180 ry 0 rz -180 deg; joints [3.26, 68.813, -33.313, 5.601, -35.629, -4.558]
  Call Extruder -0.32834
  MoveL (T17542) to (103.65, 102.72, 18.9) mm, rotated rx 180 ry 0 rz -180 deg; joints [3.26, 68.813, -33.313, 5.601, -35.629, -4.558]
  Set speed (45.0 mm/s)
  Call Extruder -0.02
  MoveL (T17543) to (103.65, 102.72, 18.9) mm, rotated rx 180 ry 0 rz -180 deg; joints [2.685, 70.244, -36.003, 4.764, -34.334, -3.936]
  Set speed (150.0 mm/s)
  MoveL (T17544) to (103.65, 102.72, 20.9) mm, rotated rx 180 ry 0 rz -180 deg; joints [2.754, 70.464, -36.415, 4.911, -34.146, -4.067]
  MoveL (T17545) to (117.73, 104.5, 20.9) mm, rotated rx 180 ry 0 rz -180 deg; joints [2.754, 70.464, -36.415, 4.911, -34.146, -4.067]
  MoveL (T17546) to (117.73, 104.5, 18.9) mm, rotated rx 180 ry 0 rz -180 deg; joints [2.754, 70.464, -36.415, 4.911, -34.146, -4.067]
  Set speed (40.0 mm/s)
  Call Extruder 2.0
  MoveL (T17547) to (117.73, 104.5, 18.9) mm, rotated rx 180 ry 0 rz -180 deg; joints [2.762, 70.526, -36.533, 4.931, -34.092, -4.087]
  Call Extruder 0.02918
  MoveL (T17548) to (117.07, 105.16, 18.9) mm, rotated rx 180 ry 0 rz -180 deg; joints [2.762, 70.526, -36.533, 4.931, -34.092, -4.087]
  Call Extruder 0.01841
  MoveL (T17549) to (116.48, 105.16, 18.9) mm, rotated rx 180 ry 0 rz -180 deg; joints [2.762, 70.526, -36.533, 4.931, -34.092, -4.087]
  Call Extruder 0.04713
  MoveL (T17550) to (117.55, 104.09, 18.9) mm, rotated rx 180 ry 0 rz -180 deg; joints [2.762, 70.526, -36.533, 4.931, -34.092, -4.087]
  Call Extruder 0.00782
  MoveL (T17551) to (117.55, 103.84, 18.9) mm, rotated rx 180 ry 0 rz -180 deg; joints [2.762, 70.526, -36.533, 4.931, -34.092, -4.087]
  Call Extruder 0.01059
  MoveL (T17552) to (117.21, 103.84, 18.9) mm, rotated rx 180 ry 0 rz -180 deg; joints [2.756, 70.91, -37.254, 4.964, -33.756, -4.13]
  Call Extruder 0.05818
  MoveL (T17553) to (115.89, 105.16, 18.9) mm, rotated rx 180 ry 0 rz -180 deg; joints [2.756, 70.91, -37.254, 4.964, -33.756, -4.13]
  Call Extruder 0.01841
  MoveL (T17554) to (115.3, 105.16, 18.9) mm, rotated rx 180 ry 0 rz -180 deg; joints [2.756, 70.91, -37.254, 4.964, -33.756, -4.13]
  Call Extruder 0.05818
  MoveL (T17555) to (116.62, 103.84, 18.9) mm, rotated rx 180 ry 0 rz -180 deg; joints [2.756, 70.91, -37.254, 4.964, -33.756, -4.13]
  Call Extruder 0.01841
  MoveL (T17556) to (116.03, 103.84, 18.9) mm, rotated rx 180 ry 0 rz -180 deg; joints [2.756, 70.91, -37.254, 4.964, -33.756, -4.13]
  Call Extruder 0.05818
  MoveL (T17557) to (114.71, 105.16, 18.9) mm, rotated rx 180 ry 0 rz -180 deg; joints [2.756, 70.91, -37.254, 4.964, -33.756, -4.13]
  Call Extruder 0.01841
  MoveL (T17558) to (114.12, 105.16, 18.9) mm, rotated rx 180 ry 0 rz -180 deg; joints [2.756, 70.91, -37.254, 4.964, -33.756, -4.13]
  Call Extruder 0.05818
  MoveL (T17559) to (115.44, 103.84, 18.9) mm, rotated rx 180 ry 0 rz -180 deg; joints [2.756, 70.91, -37.254, 4.964, -33.756, -4.13]
  Call Extruder 0.01841
  MoveL (T17560) to (114.85, 103.84, 18.9) mm, rotated rx 180 ry 0 rz -180 deg; joints [2.761, 70.581, -36.636, 4.936, -34.044, -4.093]
  Call Extruder 0.05818
  MoveL (T17561) to (113.53, 105.16, 18.9) mm, rotated rx 180 ry 0 rz -180 deg; joints [2.761, 70.581, -36.636, 4.936, -34.044, -4.093]
  Call Extruder 0.01841
  MoveL (T17562) to (112.94, 105.16, 18.9) mm, rotated rx 180 ry 0 rz -180 deg; joints [2.761, 70.581, -36.636, 4.936, -34.044, -4.093]
  Call Extruder 0.05818
  MoveL (T17563) to (114.26, 103.84, 18.9) mm, rotated rx 180 ry 0 rz -180 deg; joints [2.761, 70.581, -36.636, 4.936, -34.044, -4.093]
  Call Extruder 0.01841
  MoveL (T17564) to (113.67, 103.84, 18.9) mm, rotated rx 180 ry 0 rz -180 deg; joints [2.761, 70.581, -36.636, 4.936, -34.044, -4.093]
  Call Extruder 0.05818
  MoveL (T17565) to (112.35, 105.16, 18.9) mm, rotated rx 180 ry 0 rz -180 deg; joints [2.761, 70.581, -36.636, 4.936, -34.044, -4.093]
  Call Extruder 0.01841
  MoveL (T17566) to (111.76, 105.16, 18.9) mm, rotated rx 180 ry 0 rz -180 deg; joints [2.761, 70.581, -36.636, 4.936, -34.044, -4.093]
  Call Extruder 0.05818
  MoveL (T17567) to (113.08, 103.84, 18.9) mm, rotated rx 180 ry 0 rz -180 deg; joints [2.761, 70.581, -36.636, 4.936, -34.044, -4.093]
  Call Extruder 0.01841
  MoveL (T17568) to (112.49, 103.84, 18.9) mm, rotated rx 180 ry 0 rz -180 deg; joints [2.761, 70.581, -36.636, 4.936, -34.044, -4.093]
  Call Extruder 0.05818
  MoveL (T17569) to (111.17, 105.16, 18.9) mm, rotated rx 180 ry 0 rz -180 deg; joints [2.761, 70.348, -36.594, 4.961, -33.854, -4.123]
  Call Extruder 0.01841
  MoveL (T17570) to (110.58, 105.16, 18.9) mm, rotated rx 180 ry 0 rz -180 deg; joints [1.813, 70.591, -37.05, 3.278, -33.585, -2.732]
  Call Extruder 0.05818
  MoveL (T17571) to (111.9, 103.84, 18.9) mm, rotated rx 180 ry 0 rz -180 deg; joints [1.813, 70.824, -37.092, 3.262, -33.775, -2.712]
  Call Extruder 0.01841
  MoveL (T17572) to (111.31, 103.84, 18.9) mm, rotated rx 180 ry 0 rz -180 deg; joints [1.813, 70.824, -37.092, 3.262, -33.775, -2.712]
  Call Extruder 0.05818
  MoveL (T17573) to (109.99, 105.16, 18.9) mm, rotated rx 180 ry 0 rz -180 deg; joints [1.813, 70.824, -37.092, 3.262, -33.775, -2.712]
  Call Extruder 0.01841
  MoveL (T17574) to (109.4, 105.16, 18.9) mm, rotated rx 180 ry 0 rz -180 deg; joints [1.813, 70.824, -37.092, 3.262, -33.775, -2.712]
  Call Extruder 0.05818
  MoveL (T17575) to (110.72, 103.84, 18.9) mm, rotated rx 180 ry 0 rz -180 deg; joints [1.813, 70.824, -37.092, 3.262, -33.775, -2.712]
  Call Extruder 0.01841
  MoveL (T17576) to (110.13, 103.84, 18.9) mm, rotated rx 180 ry 0 rz -180 deg; joints [1.813, 70.824, -37.092, 3.262, -33.775, -2.712]
  Call Extruder 0.05818
  MoveL (T17577) to (108.81, 105.16, 18.9) mm, rotated rx 180 ry 0 rz -180 deg; joints [1.813, 70.824, -37.092, 3.262, -33.775, -2.712]
  Call Extruder 0.01841
  MoveL (T17578) to (108.22, 105.16, 18.9) mm, rotated rx 180 ry 0 rz -180 deg; joints [1.813, 70.824, -37.092, 3.262, -33.775, -2.712]
  Call Extruder 0.05818
  MoveL (T17579) to (109.54, 103.84, 18.9) mm, rotated rx 180 ry 0 rz -180 deg; joints [1.813, 70.824, -37.092, 3.262, -33.775, -2.712]
  Call Extruder 0.01841
  MoveL (T17580) to (108.95, 103.84, 18.9) mm, rotated rx 180 ry 0 rz -180 deg; joints [1.813, 70.824, -37.092, 3.262, -33.775, -2.712]
  Call Extruder 0.04712
  MoveL (T17581) to (107.89, 104.91, 18.9) mm, rotated rx 180 ry 0 rz -180 deg; joints [1.813, 70.824, -37.092, 3.262, -33.775, -2.712]
  Call Extruder 0.01841
  MoveL (T17582) to (107.89, 104.32, 18.9) mm, rotated rx 180 ry 0 rz -180 deg; joints [1.886, 71.054, -37.525, 3.411, -33.576, -2.843]
  Call Extruder 0.02917
  MoveL (T17583) to (108.55, 103.66, 18.9) mm, rotated rx 180 ry 0 rz -180 deg; joints [1.886, 71.054, -37.525, 3.411, -33.576, -2.843]
  Set speed (45.0 mm/s)
  Call Extruder -1.6
  MoveL (T17584) to (108.55, 103.66, 18.9) mm, rotated rx 180 ry 0 rz -180 deg; joints [1.886, 71.054, -37.525, 3.411, -33.576, -2.843]
  Set speed (120.0 mm/s)
  MoveL (T17585) to (108.55, 103.66, 18.9) mm, rotated rx 180 ry 0 rz -180 deg; joints [1.946, 71.06, -37.536, 3.521, -33.574, -2.935]
  Call Extruder -0.33294
  MoveL (T17586) to (107.89, 104.32, 18.9) mm, rotated rx 180 ry 0 rz -180 deg; joints [1.946, 71.06, -37.536, 3.521, -33.574, -2.935]
  Call Extruder -0.04706
  MoveL (T17587) to (107.89, 104.45, 18.9) mm, rotated rx 180 ry 0 rz -180 deg; joints [1.946, 71.06, -37.536, 3.521, -33.574, -2.935]
  Set speed (45.0 mm/s)
  Call Extruder -0.02
  MoveL (T17588) to (107.89, 104.45, 18.9) mm, rotated rx 180 ry 0 rz -180 deg; joints [1.833, 70.703, -36.865, 3.29, -33.882, -2.732]
  Set speed (150.0 mm/s)
  MoveL (T17589) to (107.89, 104.45, 20.9) mm, rotated rx 180 ry 0 rz -180 deg; joints [1.833, 70.703, -36.865, 3.29, -33.882, -2.732]
  MoveL (T17590) to (111.74, 116.15, 20.9) mm, rotated rx 180 ry 0 rz -180 deg; joints [1.835, 70.526, -36.532, 3.28, -34.038, -2.719]
  MoveL (T17591) to (111.74, 116.15, 18.9) mm, rotated rx 180 ry 0 rz -180 deg; joints [1.835, 70.526, -36.532, 3.28, -34.038, -2.719]
  Set speed (40.0 mm/s)
  Call Extruder 2.0
  MoveL (T17592) to (111.74, 116.15, 18.9) mm, rotated rx 180 ry 0 rz -180 deg; joints [2.007, 71.066, -37.548, 3.631, -33.572, -3.027]
  Set speed (25.0 mm/s)
  MoveL (T17593) to (111.74, 116.15, 18.9) mm, rotated rx 180 ry 0 rz -180 deg; joints [2.007, 71.066, -37.548, 3.631, -33.572, -3.027]
  Call Extruder 0.00774
  MoveL (T17594) to (111.94, 115.94, 18.9) mm, rotated rx 180 ry 0 rz -180 deg; joints [2.007, 71.066, -37.548, 3.631, -33.572, -3.027]
  Call Extruder 0.00969
